Staubli VAL3: sad_proj_sin.dtx

public frame fReference = {x=1365.054, y=-125.975, z=-1150, rz=90, fatherId=world[0]}
public jointRx jPark = {j3=90, j5=90}
public jointRx jJoint = {j1=-39.51779, j2=74.82624, j3=56.29695, j5=48.87681, j6=-167.66375}
public mdesc mNomSpeed = {tmax=100, rmax=100, leave=0.1, reach=0.1, blend=cartesian}
public pointRx pPoint[4564]
  [0] = {x=-1000, z=100, rx=180, rz=141.854, shoulder=lefty, elbow=epositive, wrist=wpositive, fatherId=fReference[0]}
  [1] = {x=-1000, rx=180, rz=141.854, shoulder=lefty, elbow=epositive, wrist=wpositive, fatherId=fReference[0]}
  [2] = {x=-1000, rx=180, rz=141.854, shoulder=lefty, elbow=epositive, wrist=wpositive, fatherId=fReference[0]}
  [3] = {x=-998.763, y=0.971, rx=180, rz=141.854, shoulder=lefty, elbow=epositive, wrist=wpositive, fatherId=fReference[0]}
  [4] = {x=-997.527, y=1.942, rx=180, rz=141.855, shoulder=lefty, elbow=epositive, wrist=wpositive, fatherId=fReference[0]}
  [5] = {x=-996.29, y=2.914, rx=180, rz=141.857, shoulder=lefty, elbow=epositive, wrist=wpositive, fatherId=fReference[0]}
  [6] = {x=-995.054, y=3.885, rx=180, rz=141.858, shoulder=lefty, elbow=epositive, wrist=wpositive, fatherId=fReference[0]}
  [7] = {x=-993.817, y=4.856, rx=180, rz=141.86, shoulder=lefty, elbow=epositive, wrist=wpositive, fatherId=fReference[0]}
  [8] = {x=-992.58, y=5.827, rx=180, rz=141.863, shoulder=lefty, elbow=epositive, wrist=wpositive, fatherId=fReference[0]}
  [9] = {x=-991.344, y=6.798, rx=180, rz=141.866, shoulder=lefty, elbow=epositive, wrist=wpositive, fatherId=fReference[0]}
  [10] = {x=-990.107, y=7.769, rx=180, rz=141.869, shoulder=lefty, elbow=epositive, wrist=wpositive, fatherId=fReference[0]}
  [11] = {x=-988.87, y=8.739, rx=180, rz=141.873, shoulder=lefty, elbow=epositive, wrist=wpositive, fatherId=fReference[0]}
  [12] = {x=-987.634, y=9.71, rx=180, rz=141.877, shoulder=lefty, elbow=epositive, wrist=wpositive, fatherId=fReference[0]}
  [13] = {x=-986.397, y=10.681, rx=180, rz=141.882, shoulder=lefty, elbow=epositive, wrist=wpositive, fatherId=fReference[0]}
  [14] = {x=-985.16, y=11.651, rx=180, rz=141.887, shoulder=lefty, elbow=epositive, wrist=wpositive, fatherId=fReference[0]}
  [15] = {x=-983.923, y=12.622, rx=180, rz=141.892, shoulder=lefty, elbow=epositive, wrist=wpositive, fatherId=fReference[0]}
  [16] = {x=-982.686, y=13.592, rx=180, rz=141.898, shoulder=lefty, elbow=epositive, wrist=wpositive, fatherId=fReference[0]}
  [17] = {x=-981.449, y=14.562, rx=180, rz=141.904, shoulder=lefty, elbow=epositive, wrist=wpositive, fatherId=fReference[0]}
  [18] = {x=-980.211, y=15.532, rx=180, rz=141.911, shoulder=lefty, elbow=epositive, wrist=wpositive, fatherId=fReference[0]}
  [19] = {x=-978.974, y=16.502, rx=180, rz=141.918, shoulder=lefty, elbow=epositive, wrist=wpositive, fatherId=fReference[0]}
  [20] = {x=-977.737, y=17.471, rx=180, rz=141.926, shoulder=lefty, elbow=epositive, wrist=wpositive, fatherId=fReference[0]}
  [21] = {x=-976.499, y=18.441, rx=180, rz=141.934, shoulder=lefty, elbow=epositive, wrist=wpositive, fatherId=fReference[0]}
  [22] = {x=-975.262, y=19.41, rx=180, rz=141.942, shoulder=lefty, elbow=epositive, wrist=wpositive, fatherId=fReference[0]}
  [23] = {x=-974.024, y=20.379, rx=180, rz=141.951, shoulder=lefty, elbow=epositive, wrist=wpositive, fatherId=fReference[0]}
  [24] = {x=-972.786, y=21.347, rx=180, rz=141.96, shoulder=lefty, elbow=epositive, wrist=wpositive, fatherId=fReference[0]}
  [25] = {x=-971.549, y=22.316, rx=180, rz=141.97, shoulder=lefty, elbow=epositive, wrist=wpositive, fatherId=fReference[0]}
  [26] = {x=-970.311, y=23.284, rx=180, rz=141.98, shoulder=lefty, elbow=epositive, wrist=wpositive, fatherId=fReference[0]}
  [27] = {x=-969.072, y=24.252, rx=180, rz=141.991, shoulder=lefty, elbow=epositive, wrist=wpositive, fatherId=fReference[0]}
  [28] = {x=-967.834, y=25.22, rx=180, rz=142.002, shoulder=lefty, elbow=epositive, wrist=wpositive, fatherId=fReference[0]}
  [29] = {x=-966.596, y=26.187, rx=180, rz=142.013, shoulder=lefty, elbow=epositive, wrist=wpositive, fatherId=fReference[0]}
  [30] = {x=-965.357, y=27.155, rx=180, rz=142.025, shoulder=lefty, elbow=epositive, wrist=wpositive, fatherId=fReference[0]}
  [31] = {x=-964.119, y=28.121, rx=180, rz=142.037, shoulder=lefty, elbow=epositive, wrist=wpositive, fatherId=fReference[0]}
  [32] = {x=-962.88, y=29.088, rx=180, rz=142.05, shoulder=lefty, elbow=epositive, wrist=wpositive, fatherId=fReference[0]}
  [33] = {x=-961.641, y=30.054, rx=180, rz=142.063, shoulder=lefty, elbow=epositive, wrist=wpositive, fatherId=fReference[0]}
  [34] = {x=-960.402, y=31.02, rx=180, rz=142.076, shoulder=lefty, elbow=epositive, wrist=wpositive, fatherId=fReference[0]}
  [35] = {x=-959.163, y=31.986, rx=180, rz=142.09, shoulder=lefty, elbow=epositive, wrist=wpositive, fatherId=fReference[0]}
  [36] = {x=-957.923, y=32.951, rx=180, rz=142.105, shoulder=lefty, elbow=epositive, wrist=wpositive, fatherId=fReference[0]}
  [37] = {x=-956.684, y=33.916, rx=180, rz=142.12, shoulder=lefty, elbow=epositive, wrist=wpositive, fatherId=fReference[0]}
  [38] = {x=-955.444, y=34.88, rx=180, rz=142.135, shoulder=lefty, elbow=epositive, wrist=wpositive, fatherId=fReference[0]}
  [39] = {x=-954.204, y=35.844, rx=180, rz=142.151, shoulder=lefty, elbow=epositive, wrist=wpositive, fatherId=fReference[0]}
  [40] = {x=-952.964, y=36.808, rx=180, rz=142.167, shoulder=lefty, elbow=epositive, wrist=wpositive, fatherId=fReference[0]}
  [41] = {x=-951.724, y=37.771, rx=180, rz=142.183, shoulder=lefty, elbow=epositive, wrist=wpositive, fatherId=fReference[0]}
  [42] = {x=-950.483, y=38.734, rx=180, rz=142.2, shoulder=lefty, elbow=epositive, wrist=wpositive, fatherId=fReference[0]}
  [43] = {x=-949.243, y=39.696, rx=180, rz=142.218, shoulder=lefty, elbow=epositive, wrist=wpositive, fatherId=fReference[0]}
  [44] = {x=-948.002, y=40.658, rx=180, rz=142.235, shoulder=lefty, elbow=epositive, wrist=wpositive, fatherId=fReference[0]}
  [45] = {x=-946.761, y=41.619, rx=180, rz=142.254, shoulder=lefty, elbow=epositive, wrist=wpositive, fatherId=fReference[0]}
  [46] = {x=-945.52, y=42.58, rx=180, rz=142.272, shoulder=lefty, elbow=epositive, wrist=wpositive, fatherId=fReference[0]}
  [47] = {x=-944.278, y=43.541, rx=180, rz=142.291, shoulder=lefty, elbow=epositive, wrist=wpositive, fatherId=fReference[0]}
  [48] = {x=-943.037, y=44.501, rx=180, rz=142.311, shoulder=lefty, elbow=epositive, wrist=wpositive, fatherId=fReference[0]}
  [49] = {x=-941.795, y=45.46, rx=180, rz=142.331, shoulder=lefty, elbow=epositive, wrist=wpositive, fatherId=fReference[0]}
  [50] = {x=-940.553, y=46.419, rx=180, rz=142.351, shoulder=lefty, elbow=epositive, wrist=wpositive, fatherId=fReference[0]}
  [51] = {x=-939.31, y=47.377, rx=180, rz=142.372, shoulder=lefty, elbow=epositive, wrist=wpositive, fatherId=fReference[0]}
  [52] = {x=-938.068, y=48.335, rx=180, rz=142.394, shoulder=lefty, elbow=epositive, wrist=wpositive, fatherId=fReference[0]}
  [53] = {x=-936.825, y=49.292, rx=180, rz=142.415, shoulder=lefty, elbow=epositive, wrist=wpositive, fatherId=fReference[0]}
  [54] = {x=-935.582, y=50.249, rx=180, rz=142.438, shoulder=lefty, elbow=epositive, wrist=wpositive, fatherId=fReference[0]}
  [55] = {x=-934.339, y=51.205, rx=180, rz=142.46, shoulder=lefty, elbow=epositive, wrist=wpositive, fatherId=fReference[0]}
  [56] = {x=-933.095, y=52.161, rx=180, rz=142.483, shoulder=lefty, elbow=epositive, wrist=wpositive, fatherId=fReference[0]}
  [57] = {x=-931.852, y=53.116, rx=180, rz=142.507, shoulder=lefty, elbow=epositive, wrist=wpositive, fatherId=fReference[0]}
  [58] = {x=-930.608, y=54.07, rx=180, rz=142.531, shoulder=lefty, elbow=epositive, wrist=wpositive, fatherId=fReference[0]}
  [59] = {x=-929.363, y=55.024, rx=180, rz=142.555, shoulder=lefty, elbow=epositive, wrist=wpositive, fatherId=fReference[0]}
  [60] = {x=-928.119, y=55.977, rx=180, rz=142.58, shoulder=lefty, elbow=epositive, wrist=wpositive, fatherId=fReference[0]}
  [61] = {x=-926.874, y=56.929, rx=180, rz=142.605, shoulder=lefty, elbow=epositive, wrist=wpositive, fatherId=fReference[0]}
  [62] = {x=-925.629, y=57.881, rx=180, rz=142.631, shoulder=lefty, elbow=epositive, wrist=wpositive, fatherId=fReference[0]}
  [63] = {x=-924.384, y=58.832, rx=180, rz=142.657, shoulder=lefty, elbow=epositive, wrist=wpositive, fatherId=fReference[0]}
  [64] = {x=-923.138, y=59.782, rx=180, rz=142.684, shoulder=lefty, elbow=epositive, wrist=wpositive, fatherId=fReference[0]}
  [65] = {x=-921.892, y=60.732, rx=180, rz=142.711, shoulder=lefty, elbow=epositive, wrist=wpositive, fatherId=fReference[0]}
  [66] = {x=-920.646, y=61.681, rx=180, rz=142.738, shoulder=lefty, elbow=epositive, wrist=wpositive, fatherId=fReference[0]}
  [67] = {x=-919.4, y=62.629, rx=180, rz=142.766, shoulder=lefty, elbow=epositive, wrist=wpositive, fatherId=fReference[0]}
  [68] = {x=-918.153, y=63.576, rx=180, rz=142.795, shoulder=lefty, elbow=epositive, wrist=wpositive, fatherId=fReference[0]}
  [69] = {x=-916.906, y=64.523, rx=180, rz=142.824, shoulder=lefty, elbow=epositive, wrist=wpositive, fatherId=fReference[0]}
  [70] = {x=-915.659, y=65.469, rx=180, rz=142.853, shoulder=lefty, elbow=epositive, wrist=wpositive, fatherId=fReference[0]}
  [71] = {x=-914.411, y=66.414, rx=180, rz=142.883, shoulder=lefty, elbow=epositive, wrist=wpositive, fatherId=fReference[0]}
  [72] = {x=-913.163, y=67.358, rx=180, rz=142.913, shoulder=lefty, elbow=epositive, wrist=wpositive, fatherId=fReference[0]}
  [73] = {x=-911.915, y=68.302, rx=180, rz=142.944, shoulder=lefty, elbow=epositive, wrist=wpositive, fatherId=fReference[0]}
  [74] = {x=-910.667, y=69.245, rx=180, rz=142.975, shoulder=lefty, elbow=epositive, wrist=wpositive, fatherId=fReference[0]}
  [75] = {x=-909.418, y=70.187, rx=180, rz=143.007, shoulder=lefty, elbow=epositive, wrist=wpositive, fatherId=fReference[0]}
  [76] = {x=-908.169, y=71.128, rx=180, rz=143.039, shoulder=lefty, elbow=epositive, wrist=wpositive, fatherId=fReference[0]}
  [77] = {x=-906.919, y=72.068, rx=180, rz=143.071, shoulder=lefty, elbow=epositive, wrist=wpositive, fatherId=fReference[0]}
  [78] = {x=-905.67, y=73.007, rx=180, rz=143.104, shoulder=lefty, elbow=epositive, wrist=wpositive, fatherId=fReference[0]}
  [79] = {x=-904.419, y=73.946, rx=180, rz=143.138, shoulder=lefty, elbow=epositive, wrist=wpositive, fatherId=fReference[0]}
  [80] = {x=-903.169, y=74.883, rx=180, rz=143.172, shoulder=lefty, elbow=epositive, wrist=wpositive, fatherId=fReference[0]}
  [81] = {x=-901.918, y=75.82, rx=180, rz=143.206, shoulder=lefty, elbow=epositive, wrist=wpositive, fatherId=fReference[0]}
  [82] = {x=-900.667, y=76.756, rx=180, rz=143.241, shoulder=lefty, elbow=epositive, wrist=wpositive, fatherId=fReference[0]}
  [83] = {x=-899.416, y=77.691, rx=180, rz=143.276, shoulder=lefty, elbow=epositive, wrist=wpositive, fatherId=fReference[0]}
  [84] = {x=-898.164, y=78.625, rx=180, rz=143.312, shoulder=lefty, elbow=epositive, wrist=wpositive, fatherId=fReference[0]}
  [85] = {x=-896.912, y=79.557, rx=180, rz=143.348, shoulder=lefty, elbow=epositive, wrist=wpositive, fatherId=fReference[0]}
  [86] = {x=-895.659, y=80.489, rx=180, rz=143.385, shoulder=lefty, elbow=epositive, wrist=wpositive, fatherId=fReference[0]}
  [87] = {x=-894.406, y=81.42, rx=180, rz=143.422, shoulder=lefty, elbow=epositive, wrist=wpositive, fatherId=fReference[0]}
  [88] = {x=-893.153, y=82.35, rx=180, rz=143.46, shoulder=lefty, elbow=epositive, wrist=wpositive, fatherId=fReference[0]}
  [89] = {x=-891.899, y=83.279, rx=180, rz=143.498, shoulder=lefty, elbow=epositive, wrist=wpositive, fatherId=fReference[0]}
  [90] = {x=-890.645, y=84.207, rx=180, rz=143.536, shoulder=lefty, elbow=epositive, wrist=wpositive, fatherId=fReference[0]}
  [91] = {x=-889.391, y=85.134, rx=180, rz=143.575, shoulder=lefty, elbow=epositive, wrist=wpositive, fatherId=fReference[0]}
  [92] = {x=-888.136, y=86.06, rx=180, rz=143.615, shoulder=lefty, elbow=epositive, wrist=wpositive, fatherId=fReference[0]}
  [93] = {x=-886.881, y=86.985, rx=180, rz=143.655, shoulder=lefty, elbow=epositive, wrist=wpositive, fatherId=fReference[0]}
  [94] = {x=-885.626, y=87.909, rx=180, rz=143.696, shoulder=lefty, elbow=epositive, wrist=wpositive, fatherId=fReference[0]}
  [95] = {x=-884.37, y=88.832, rx=180, rz=143.737, shoulder=lefty, elbow=epositive, wrist=wpositive, fatherId=fReference[0]}
  [96] = {x=-883.113, y=89.753, rx=180, rz=143.778, shoulder=lefty, elbow=epositive, wrist=wpositive, fatherId=fReference[0]}
  [97] = {x=-881.857, y=90.674, rx=180, rz=143.82, shoulder=lefty, elbow=epositive, wrist=wpositive, fatherId=fReference[0]}
  [98] = {x=-880.6, y=91.593, rx=180, rz=143.862, shoulder=lefty, elbow=epositive, wrist=wpositive, fatherId=fReference[0]}
  [99] = {x=-879.342, y=92.511, rx=180, rz=143.905, shoulder=lefty, elbow=epositive, wrist=wpositive, fatherId=fReference[0]}
  [100] = {x=-878.084, y=93.428, rx=180, rz=143.949, shoulder=lefty, elbow=epositive, wrist=wpositive, fatherId=fReference[0]}
  [101] = {x=-876.826, y=94.344, rx=180, rz=143.993, shoulder=lefty, elbow=epositive, wrist=wpositive, fatherId=fReference[0]}
  [102] = {x=-875.567, y=95.259, rx=180, rz=144.037, shoulder=lefty, elbow=epositive, wrist=wpositive, fatherId=fReference[0]}
  [103] = {x=-874.308, y=96.173, rx=180, rz=144.082, shoulder=lefty, elbow=epositive, wrist=wpositive, fatherId=fReference[0]}
  [104] = {x=-873.049, y=97.085, rx=180, rz=144.127, shoulder=lefty, elbow=epositive, wrist=wpositive, fatherId=fReference[0]}
  [105] = {x=-871.789, y=97.996, rx=180, rz=144.173, shoulder=lefty, elbow=epositive, wrist=wpositive, fatherId=fReference[0]}
  [106] = {x=-870.528, y=98.906, rx=180, rz=144.22, shoulder=lefty, elbow=epositive, wrist=wpositive, fatherId=fReference[0]}
  [107] = {x=-869.267, y=99.815, rx=180, rz=144.266, shoulder=lefty, elbow=epositive, wrist=wpositive, fatherId=fReference[0]}
  [108] = {x=-868.006, y=100.722, rx=180, rz=144.314, shoulder=lefty, elbow=epositive, wrist=wpositive, fatherId=fReference[0]}
  [109] = {x=-866.745, y=101.628, rx=180, rz=144.362, shoulder=lefty, elbow=epositive, wrist=wpositive, fatherId=fReference[0]}
  [110] = {x=-865.482, y=102.533, rx=180, rz=144.41, shoulder=lefty, elbow=epositive, wrist=wpositive, fatherId=fReference[0]}
  [111] = {x=-864.22, y=103.437, rx=180, rz=144.459, shoulder=lefty, elbow=epositive, wrist=wpositive, fatherId=fReference[0]}
  [112] = {x=-862.957, y=104.339, rx=180, rz=144.508, shoulder=lefty, elbow=epositive, wrist=wpositive, fatherId=fReference[0]}
  [113] = {x=-861.693, y=105.24, rx=180, rz=144.558, shoulder=lefty, elbow=epositive, wrist=wpositive, fatherId=fReference[0]}
  [114] = {x=-860.429, y=106.139, rx=180, rz=144.609, shoulder=lefty, elbow=epositive, wrist=wpositive, fatherId=fReference[0]}
  [115] = {x=-859.165, y=107.038, rx=180, rz=144.659, shoulder=lefty, elbow=epositive, wrist=wpositive, fatherId=fReference[0]}
  [116] = {x=-857.9, y=107.935, rx=180, rz=144.711, shoulder=lefty, elbow=epositive, wrist=wpositive, fatherId=fReference[0]}
  [117] = {x=-856.635, y=108.83, rx=180, rz=144.763, shoulder=lefty, elbow=epositive, wrist=wpositive, fatherId=fReference[0]}
  [118] = {x=-855.369, y=109.724, rx=180, rz=144.815, shoulder=lefty, elbow=epositive, wrist=wpositive, fatherId=fReference[0]}
  [119] = {x=-854.103, y=110.617, rx=180, rz=144.868, shoulder=lefty, elbow=epositive, wrist=wpositive, fatherId=fReference[0]}
  [120] = {x=-852.836, y=111.508, rx=180, rz=144.922, shoulder=lefty, elbow=epositive, wrist=wpositive, fatherId=fReference[0]}
  [121] = {x=-851.569, y=112.398, rx=180, rz=144.976, shoulder=lefty, elbow=epositive, wrist=wpositive, fatherId=fReference[0]}
  [122] = {x=-850.301, y=113.287, rx=180, rz=145.03, shoulder=lefty, elbow=epositive, wrist=wpositive, fatherId=fReference[0]}
  [123] = {x=-849.033, y=114.174, rx=180, rz=145.085, shoulder=lefty, elbow=epositive, wrist=wpositive, fatherId=fReference[0]}
  [124] = {x=-847.764, y=115.059, rx=180, rz=145.141, shoulder=lefty, elbow=epositive, wrist=wpositive, fatherId=fReference[0]}
  [125] = {x=-846.495, y=115.943, rx=180, rz=145.197, shoulder=lefty, elbow=epositive, wrist=wpositive, fatherId=fReference[0]}
  [126] = {x=-845.225, y=116.826, rx=180, rz=145.253, shoulder=lefty, elbow=epositive, wrist=wpositive, fatherId=fReference[0]}
  [127] = {x=-843.955, y=117.707, rx=180, rz=145.311, shoulder=lefty, elbow=epositive, wrist=wpositive, fatherId=fReference[0]}
  [128] = {x=-842.685, y=118.586, rx=180, rz=145.368, shoulder=lefty, elbow=epositive, wrist=wpositive, fatherId=fReference[0]}
  [129] = {x=-841.413, y=119.464, rx=-180, rz=145.426, shoulder=lefty, elbow=epositive, wrist=wpositive, fatherId=fReference[0]}
  [130] = {x=-840.142, y=120.341, rx=180, rz=145.485, shoulder=lefty, elbow=epositive, wrist=wpositive, fatherId=fReference[0]}
  [131] = {x=-838.869, y=121.216, rx=180, rz=145.544, shoulder=lefty, elbow=epositive, wrist=wpositive, fatherId=fReference[0]}
  [132] = {x=-837.597, y=122.089, rx=180, rz=145.604, shoulder=lefty, elbow=epositive, wrist=wpositive, fatherId=fReference[0]}
  [133] = {x=-836.323, y=122.961, rx=180, rz=145.665, shoulder=lefty, elbow=epositive, wrist=wpositive, fatherId=fReference[0]}
  [134] = {x=-835.049, y=123.831, rx=180, rz=145.725, shoulder=lefty, elbow=epositive, wrist=wpositive, fatherId=fReference[0]}
  [135] = {x=-833.775, y=124.699, rx=180, rz=145.787, shoulder=lefty, elbow=epositive, wrist=wpositive, fatherId=fReference[0]}
  [136] = {x=-832.5, y=125.566, rx=180, rz=145.849, shoulder=lefty, elbow=epositive, wrist=wpositive, fatherId=fReference[0]}
  [137] = {x=-831.225, y=126.431, rx=180, rz=145.911, shoulder=lefty, elbow=epositive, wrist=wpositive, fatherId=fReference[0]}
  [138] = {x=-829.949, y=127.295, rx=180, rz=145.974, shoulder=lefty, elbow=epositive, wrist=wpositive, fatherId=fReference[0]}
  [139] = {x=-828.672, y=128.157, rx=180, rz=146.038, shoulder=lefty, elbow=epositive, wrist=wpositive, fatherId=fReference[0]}
  [140] = {x=-827.395, y=129.017, rx=180, rz=146.102, shoulder=lefty, elbow=epositive, wrist=wpositive, fatherId=fReference[0]}
  [141] = {x=-826.117, y=129.876, rx=180, rz=146.167, shoulder=lefty, elbow=epositive, wrist=wpositive, fatherId=fReference[0]}
  [142] = {x=-824.839, y=130.732, rx=180, rz=146.232, shoulder=lefty, elbow=epositive, wrist=wpositive, fatherId=fReference[0]}
  [143] = {x=-823.56, y=131.587, rx=180, rz=146.298, shoulder=lefty, elbow=epositive, wrist=wpositive, fatherId=fReference[0]}
  [144] = {x=-822.281, y=132.441, rx=180, rz=146.364, shoulder=lefty, elbow=epositive, wrist=wpositive, fatherId=fReference[0]}
  [145] = {x=-821.001, y=133.292, rx=180, rz=146.431, shoulder=lefty, elbow=epositive, wrist=wpositive, fatherId=fReference[0]}
  [146] = {x=-819.721, y=134.142, rx=180, rz=146.499, shoulder=lefty, elbow=epositive, wrist=wpositive, fatherId=fReference[0]}
  [147] = {x=-818.44, y=134.99, rx=180, rz=146.567, shoulder=lefty, elbow=epositive, wrist=wpositive, fatherId=fReference[0]}
  [148] = {x=-817.158, y=135.836, rx=180, rz=146.636, shoulder=lefty, elbow=epositive, wrist=wpositive, fatherId=fReference[0]}
  [149] = {x=-815.876, y=136.68, rx=180, rz=146.705, shoulder=lefty, elbow=epositive, wrist=wpositive, fatherId=fReference[0]}
  [150] = {x=-814.593, y=137.523, rx=180, rz=146.775, shoulder=lefty, elbow=epositive, wrist=wpositive, fatherId=fReference[0]}
  [151] = {x=-813.309, y=138.364, rx=180, rz=146.845, shoulder=lefty, elbow=epositive, wrist=wpositive, fatherId=fReference[0]}
  [152] = {x=-812.025, y=139.202, rx=180, rz=146.916, shoulder=lefty, elbow=epositive, wrist=wpositive, fatherId=fReference[0]}
  [153] = {x=-810.74, y=140.039, rx=180, rz=146.987, shoulder=lefty, elbow=epositive, wrist=wpositive, fatherId=fReference[0]}
  [154] = {x=-809.455, y=140.875, rx=180, rz=147.059, shoulder=lefty, elbow=epositive, wrist=wpositive, fatherId=fReference[0]}
  [155] = {x=-808.169, y=141.708, rx=180, rz=147.132, shoulder=lefty, elbow=epositive, wrist=wpositive, fatherId=fReference[0]}
  [156] = {x=-806.883, y=142.539, rx=180, rz=147.205, shoulder=lefty, elbow=epositive, wrist=wpositive, fatherId=fReference[0]}
  [157] = {x=-805.596, y=143.368, rx=180, rz=147.279, shoulder=lefty, elbow=epositive, wrist=wpositive, fatherId=fReference[0]}
  [158] = {x=-804.308, y=144.196, rx=180, rz=147.353, shoulder=lefty, elbow=epositive, wrist=wpositive, fatherId=fReference[0]}
  [159] = {x=-803.019, y=145.021, rx=180, rz=147.428, shoulder=lefty, elbow=epositive, wrist=wpositive, fatherId=fReference[0]}
  [160] = {x=-801.73, y=145.845, rx=180, rz=147.504, shoulder=lefty, elbow=epositive, wrist=wpositive, fatherId=fReference[0]}
  [161] = {x=-800.44, y=146.666, rx=180, rz=147.58, shoulder=lefty, elbow=epositive, wrist=wpositive, fatherId=fReference[0]}
  [162] = {x=-799.15, y=147.486, rx=180, rz=147.657, shoulder=lefty, elbow=epositive, wrist=wpositive, fatherId=fReference[0]}
  [163] = {x=-797.859, y=148.303, rx=180, rz=147.734, shoulder=lefty, elbow=epositive, wrist=wpositive, fatherId=fReference[0]}
  [164] = {x=-796.567, y=149.119, rx=180, rz=147.812, shoulder=lefty, elbow=epositive, wrist=wpositive, fatherId=fReference[0]}
  [165] = {x=-795.275, y=149.932, rx=-180, rz=147.891, shoulder=lefty, elbow=epositive, wrist=wpositive, fatherId=fReference[0]}
  [166] = {x=-793.982, y=150.744, rx=180, rz=147.97, shoulder=lefty, elbow=epositive, wrist=wpositive, fatherId=fReference[0]}
  [167] = {x=-792.688, y=151.553, rx=180, rz=148.05, shoulder=lefty, elbow=epositive, wrist=wpositive, fatherId=fReference[0]}
  [168] = {x=-791.394, y=152.36, rx=180, rz=148.13, shoulder=lefty, elbow=epositive, wrist=wpositive, fatherId=fReference[0]}
  [169] = {x=-790.099, y=153.165, rx=180, rz=148.211, shoulder=lefty, elbow=epositive, wrist=wpositive, fatherId=fReference[0]}
  [170] = {x=-788.803, y=153.968, rx=180, rz=148.293, shoulder=lefty, elbow=epositive, wrist=wpositive, fatherId=fReference[0]}
  [171] = {x=-787.507, y=154.769, rx=180, rz=148.375, shoulder=lefty, elbow=epositive, wrist=wpositive, fatherId=fReference[0]}
  [172] = {x=-786.21, y=155.568, rx=180, rz=148.458, shoulder=lefty, elbow=epositive, wrist=wpositive, fatherId=fReference[0]}
  [173] = {x=-784.912, y=156.365, rx=-180, rz=148.541, shoulder=lefty, elbow=epositive, wrist=wpositive, fatherId=fReference[0]}
  [174] = {x=-783.613, y=157.159, rx=180, rz=148.625, shoulder=lefty, elbow=epositive, wrist=wpositive, fatherId=fReference[0]}
  [175] = {x=-782.314, y=157.951, rx=180, rz=148.71, shoulder=lefty, elbow=epositive, wrist=wpositive, fatherId=fReference[0]}
  [176] = {x=-781.014, y=158.741, rx=180, rz=148.795, shoulder=lefty, elbow=epositive, wrist=wpositive, fatherId=fReference[0]}
  [177] = {x=-779.714, y=159.529, rx=180, rz=148.881, shoulder=lefty, elbow=epositive, wrist=wpositive, fatherId=fReference[0]}
  [178] = {x=-778.413, y=160.315, rx=180, rz=148.968, shoulder=lefty, elbow=epositive, wrist=wpositive, fatherId=fReference[0]}
  [179] = {x=-777.111, y=161.098, rx=180, rz=149.055, shoulder=lefty, elbow=epositive, wrist=wpositive, fatherId=fReference[0]}
  [180] = {x=-775.808, y=161.879, rx=180, rz=149.143, shoulder=lefty, elbow=epositive, wrist=wpositive, fatherId=fReference[0]}
  [181] = {x=-774.505, y=162.658, rx=180, rz=149.231, shoulder=lefty, elbow=epositive, wrist=wpositive, fatherId=fReference[0]}
  [182] = {x=-773.2, y=163.434, rx=180, rz=149.32, shoulder=lefty, elbow=epositive, wrist=wpositive, fatherId=fReference[0]}
  [183] = {x=-771.896, y=164.208, rx=180, rz=149.41, shoulder=lefty, elbow=epositive, wrist=wpositive, fatherId=fReference[0]}
  [184] = {x=-770.59, y=164.98, rx=180, rz=149.5, shoulder=lefty, elbow=epositive, wrist=wpositive, fatherId=fReference[0]}
  [185] = {x=-769.284, y=165.75, rx=180, rz=149.591, shoulder=lefty, elbow=epositive, wrist=wpositive, fatherId=fReference[0]}
  [186] = {x=-767.977, y=166.517, rx=180, rz=149.683, shoulder=lefty, elbow=epositive, wrist=wpositive, fatherId=fReference[0]}
  [187] = {x=-766.669, y=167.281, rx=180, rz=149.775, shoulder=lefty, elbow=epositive, wrist=wpositive, fatherId=fReference[0]}
  [188] = {x=-765.36, y=168.044, rx=180, rz=149.868, shoulder=lefty, elbow=epositive, wrist=wpositive, fatherId=fReference[0]}
  [189] = {x=-764.051, y=168.804, rx=180, rz=149.962, shoulder=lefty, elbow=epositive, wrist=wpositive, fatherId=fReference[0]}
  [190] = {x=-762.741, y=169.561, rx=180, rz=150.056, shoulder=lefty, elbow=epositive, wrist=wpositive, fatherId=fReference[0]}
  [191] = {x=-761.431, y=170.316, rx=180, rz=150.151, shoulder=lefty, elbow=epositive, wrist=wpositive, fatherId=fReference[0]}
  [192] = {x=-760.119, y=171.069, rx=180, rz=150.247, shoulder=lefty, elbow=epositive, wrist=wpositive, fatherId=fReference[0]}
  [193] = {x=-758.807, y=171.819, rx=180, rz=150.343, shoulder=lefty, elbow=epositive, wrist=wpositive, fatherId=fReference[0]}
  [194] = {x=-757.494, y=172.566, rx=180, rz=150.44, shoulder=lefty, elbow=epositive, wrist=wpositive, fatherId=fReference[0]}
  [195] = {x=-756.181, y=173.311, rx=180, rz=150.537, shoulder=lefty, elbow=epositive, wrist=wpositive, fatherId=fReference[0]}
  [196] = {x=-754.866, y=174.054, rx=180, rz=150.636, shoulder=lefty, elbow=epositive, wrist=wpositive, fatherId=fReference[0]}
  [197] = {x=-753.551, y=174.794, rx=180, rz=150.734, shoulder=lefty, elbow=epositive, wrist=wpositive, fatherId=fReference[0]}
  [198] = {x=-752.235, y=175.531, rx=-180, rz=150.834, shoulder=lefty, elbow=epositive, wrist=wpositive, fatherId=fReference[0]}
  [199] = {x=-750.919, y=176.266, rx=-180, rz=150.934, shoulder=lefty, elbow=epositive, wrist=wpositive, fatherId=fReference[0]}
  [200] = {x=-749.601, y=176.998, rx=-180, rz=151.035, shoulder=lefty, elbow=epositive, wrist=wpositive, fatherId=fReference[0]}
  [201] = {x=-748.283, y=177.727, rx=180, rz=151.137, shoulder=lefty, elbow=epositive, wrist=wpositive, fatherId=fReference[0]}
  [202] = {x=-746.965, y=178.454, rx=180, rz=151.239, shoulder=lefty, elbow=epositive, wrist=wpositive, fatherId=fReference[0]}
  [203] = {x=-745.645, y=179.179, rx=180, rz=151.342, shoulder=lefty, elbow=epositive, wrist=wpositive, fatherId=fReference[0]}
  [204] = {x=-744.325, y=179.9, rx=180, rz=151.445, shoulder=lefty, elbow=epositive, wrist=wpositive, fatherId=fReference[0]}
  [205] = {x=-743.004, y=180.619, rx=180, rz=151.549, shoulder=lefty, elbow=epositive, wrist=wpositive, fatherId=fReference[0]}
  [206] = {x=-741.682, y=181.335, rx=180, rz=151.654, shoulder=lefty, elbow=epositive, wrist=wpositive, fatherId=fReference[0]}
  [207] = {x=-740.359, y=182.049, rx=180, rz=151.76, shoulder=lefty, elbow=epositive, wrist=wpositive, fatherId=fReference[0]}
  [208] = {x=-739.036, y=182.76, rx=180, rz=151.866, shoulder=lefty, elbow=epositive, wrist=wpositive, fatherId=fReference[0]}
  [209] = {x=-737.712, y=183.468, rx=180, rz=151.973, shoulder=lefty, elbow=epositive, wrist=wpositive, fatherId=fReference[0]}
  [210] = {x=-736.387, y=184.173, rx=180, rz=152.081, shoulder=lefty, elbow=epositive, wrist=wpositive, fatherId=fReference[0]}
  [211] = {x=-735.061, y=184.875, rx=180, rz=152.189, shoulder=lefty, elbow=epositive, wrist=wpositive, fatherId=fReference[0]}
  [212] = {x=-733.735, y=185.575, rx=180, rz=152.298, shoulder=lefty, elbow=epositive, wrist=wpositive, fatherId=fReference[0]}
  [213] = {x=-732.408, y=186.272, rx=180, rz=152.408, shoulder=lefty, elbow=epositive, wrist=wpositive, fatherId=fReference[0]}
  [214] = {x=-731.08, y=186.966, rx=-180, rz=152.518, shoulder=lefty, elbow=epositive, wrist=wpositive, fatherId=fReference[0]}
  [215] = {x=-729.751, y=187.657, rx=180, rz=152.63, shoulder=lefty, elbow=epositive, wrist=wpositive, fatherId=fReference[0]}
  [216] = {x=-728.422, y=188.345, rx=180, rz=152.741, shoulder=lefty, elbow=epositive, wrist=wpositive, fatherId=fReference[0]}
  [217] = {x=-727.092, y=189.03, rx=180, rz=152.854, shoulder=lefty, elbow=epositive, wrist=wpositive, fatherId=fReference[0]}
  [218] = {x=-725.761, y=189.713, rx=180, rz=152.967, shoulder=lefty, elbow=epositive, wrist=wpositive, fatherId=fReference[0]}
  [219] = {x=-724.429, y=190.392, rx=180, rz=153.081, shoulder=lefty, elbow=epositive, wrist=wpositive, fatherId=fReference[0]}
  [220] = {x=-723.097, y=191.069, rx=180, rz=153.196, shoulder=lefty, elbow=epositive, wrist=wpositive, fatherId=fReference[0]}
  [221] = {x=-721.764, y=191.742, rx=180, rz=153.311, shoulder=lefty, elbow=epositive, wrist=wpositive, fatherId=fReference[0]}
  [222] = {x=-720.43, y=192.413, rx=180, rz=153.427, shoulder=lefty, elbow=epositive, wrist=wpositive, fatherId=fReference[0]}
  [223] = {x=-719.095, y=193.08, rx=180, rz=153.544, shoulder=lefty, elbow=epositive, wrist=wpositive, fatherId=fReference[0]}
  [224] = {x=-717.76, y=193.745, rx=180, rz=153.661, shoulder=lefty, elbow=epositive, wrist=wpositive, fatherId=fReference[0]}
  [225] = {x=-716.424, y=194.406, rx=-180, rz=153.779, shoulder=lefty, elbow=epositive, wrist=wpositive, fatherId=fReference[0]}
  [226] = {x=-715.087, y=195.065, rx=180, rz=153.898, shoulder=lefty, elbow=epositive, wrist=wpositive, fatherId=fReference[0]}
  [227] = {x=-713.749, y=195.72, rx=180, rz=154.017, shoulder=lefty, elbow=epositive, wrist=wpositive, fatherId=fReference[0]}
  [228] = {x=-712.411, y=196.372, rx=180, rz=154.138, shoulder=lefty, elbow=epositive, wrist=wpositive, fatherId=fReference[0]}
  [229] = {x=-711.072, y=197.022, rx=180, rz=154.259, shoulder=lefty, elbow=epositive, wrist=wpositive, fatherId=fReference[0]}
  [230] = {x=-709.732, y=197.668, rx=180, rz=154.38, shoulder=lefty, elbow=epositive, wrist=wpositive, fatherId=fReference[0]}
  [231] = {x=-708.391, y=198.311, rx=180, rz=154.503, shoulder=lefty, elbow=epositive, wrist=wpositive, fatherId=fReference[0]}
  [232] = {x=-707.05, y=198.95, rx=180, rz=154.626, shoulder=lefty, elbow=epositive, wrist=wpositive, fatherId=fReference[0]}
  [233] = {x=-705.708, y=199.587, rx=180, rz=154.75, shoulder=lefty, elbow=epositive, wrist=wpositive, fatherId=fReference[0]}
  [234] = {x=-704.365, y=200.22, rx=-180, rz=154.874, shoulder=lefty, elbow=epositive, wrist=wpositive, fatherId=fReference[0]}
  [235] = {x=-703.021, y=200.85, rx=180, rz=154.999, shoulder=lefty, elbow=epositive, wrist=wpositive, fatherId=fReference[0]}
  [236] = {x=-701.677, y=201.477, rx=180, rz=155.125, shoulder=lefty, elbow=epositive, wrist=wpositive, fatherId=fReference[0]}
  [237] = {x=-700.332, y=202.101, rx=180, rz=155.252, shoulder=lefty, elbow=epositive, wrist=wpositive, fatherId=fReference[0]}
  [238] = {x=-698.986, y=202.721, rx=180, rz=155.379, shoulder=lefty, elbow=epositive, wrist=wpositive, fatherId=fReference[0]}
  [239] = {x=-697.639, y=203.338, rx=-180, rz=155.508, shoulder=lefty, elbow=epositive, wrist=wpositive, fatherId=fReference[0]}
  [240] = {x=-696.292, y=203.952, rx=180, rz=155.636, shoulder=lefty, elbow=epositive, wrist=wpositive, fatherId=fReference[0]}
  [241] = {x=-694.944, y=204.563, rx=180, rz=155.766, shoulder=lefty, elbow=epositive, wrist=wpositive, fatherId=fReference[0]}
  [242] = {x=-693.595, y=205.17, rx=-180, rz=155.896, shoulder=lefty, elbow=epositive, wrist=wpositive, fatherId=fReference[0]}
  [243] = {x=-692.246, y=205.774, rx=-180, rz=156.027, shoulder=lefty, elbow=epositive, wrist=wpositive, fatherId=fReference[0]}
  [244] = {x=-690.895, y=206.374, rx=180, rz=156.159, shoulder=lefty, elbow=epositive, wrist=wpositive, fatherId=fReference[0]}
  [245] = {x=-689.544, y=206.971, rx=180, rz=156.291, shoulder=lefty, elbow=epositive, wrist=wpositive, fatherId=fReference[0]}
  [246] = {x=-688.193, y=207.565, rx=180, rz=156.425, shoulder=lefty, elbow=epositive, wrist=wpositive, fatherId=fReference[0]}
  [247] = {x=-686.84, y=208.155, rx=180, rz=156.559, shoulder=lefty, elbow=epositive, wrist=wpositive, fatherId=fReference[0]}
  [248] = {x=-685.487, y=208.741, rx=180, rz=156.693, shoulder=lefty, elbow=epositive, wrist=wpositive, fatherId=fReference[0]}
  [249] = {x=-684.133, y=209.325, rx=180, rz=156.828, shoulder=lefty, elbow=epositive, wrist=wpositive, fatherId=fReference[0]}
  [250] = {x=-682.778, y=209.905, rx=180, rz=156.965, shoulder=lefty, elbow=epositive, wrist=wpositive, fatherId=fReference[0]}
  [251] = {x=-681.423, y=210.481, rx=180, rz=157.101, shoulder=lefty, elbow=epositive, wrist=wpositive, fatherId=fReference[0]}
  [252] = {x=-680.067, y=211.054, rx=180, rz=157.239, shoulder=lefty, elbow=epositive, wrist=wpositive, fatherId=fReference[0]}
  [253] = {x=-678.71, y=211.623, rx=180, rz=157.377, shoulder=lefty, elbow=epositive, wrist=wpositive, fatherId=fReference[0]}
  [254] = {x=-677.353, y=212.189, rx=180, rz=157.516, shoulder=lefty, elbow=epositive, wrist=wpositive, fatherId=fReference[0]}
  [255] = {x=-675.994, y=212.751, rx=180, rz=157.656, shoulder=lefty, elbow=epositive, wrist=wpositive, fatherId=fReference[0]}
  [256] = {x=-674.635, y=213.309, rx=180, rz=157.796, shoulder=lefty, elbow=epositive, wrist=wpositive, fatherId=fReference[0]}
  [257] = {x=-673.276, y=213.864, rx=180, rz=157.937, shoulder=lefty, elbow=epositive, wrist=wpositive, fatherId=fReference[0]}
  [258] = {x=-671.915, y=214.416, rx=180, rz=158.079, shoulder=lefty, elbow=epositive, wrist=wpositive, fatherId=fReference[0]}
  [259] = {x=-670.554, y=214.963, rx=180, rz=158.222, shoulder=lefty, elbow=epositive, wrist=wpositive, fatherId=fReference[0]}
  [260] = {x=-669.193, y=215.508, rx=180, rz=158.365, shoulder=lefty, elbow=epositive, wrist=wpositive, fatherId=fReference[0]}
  [261] = {x=-667.83, y=216.048, rx=180, rz=158.509, shoulder=lefty, elbow=epositive, wrist=wpositive, fatherId=fReference[0]}
  [262] = {x=-666.467, y=216.585, rx=180, rz=158.654, shoulder=lefty, elbow=epositive, wrist=wpositive, fatherId=fReference[0]}
  [263] = {x=-665.103, y=217.118, rx=180, rz=158.799, shoulder=lefty, elbow=epositive, wrist=wpositive, fatherId=fReference[0]}
  [264] = {x=-663.739, y=217.647, rx=180, rz=158.945, shoulder=lefty, elbow=epositive, wrist=wpositive, fatherId=fReference[0]}
  [265] = {x=-662.373, y=218.173, rx=180, rz=159.092, shoulder=lefty, elbow=epositive, wrist=wpositive, fatherId=fReference[0]}
  [266] = {x=-661.007, y=218.694, rx=180, rz=159.24, shoulder=lefty, elbow=epositive, wrist=wpositive, fatherId=fReference[0]}
  [267] = {x=-659.641, y=219.212, rx=180, rz=159.388, shoulder=lefty, elbow=epositive, wrist=wpositive, fatherId=fReference[0]}
  [268] = {x=-658.273, y=219.727, rx=180, rz=159.537, shoulder=lefty, elbow=epositive, wrist=wpositive, fatherId=fReference[0]}
  [269] = {x=-656.905, y=220.237, rx=-180, rz=159.687, shoulder=lefty, elbow=epositive, wrist=wpositive, fatherId=fReference[0]}
  [270] = {x=-655.537, y=220.744, rx=180, rz=159.837, shoulder=lefty, elbow=epositive, wrist=wpositive, fatherId=fReference[0]}
  [271] = {x=-654.167, y=221.247, rx=180, rz=159.988, shoulder=lefty, elbow=epositive, wrist=wpositive, fatherId=fReference[0]}
  [272] = {x=-652.797, y=221.746, rx=180, rz=160.14, shoulder=lefty, elbow=epositive, wrist=wpositive, fatherId=fReference[0]}
  [273] = {x=-651.426, y=222.241, rx=180, rz=160.293, shoulder=lefty, elbow=epositive, wrist=wpositive, fatherId=fReference[0]}
  [274] = {x=-650.055, y=222.732, rx=180, rz=160.446, shoulder=lefty, elbow=epositive, wrist=wpositive, fatherId=fReference[0]}
  [275] = {x=-648.683, y=223.219, rx=-180, rz=160.6, shoulder=lefty, elbow=epositive, wrist=wpositive, fatherId=fReference[0]}
  [276] = {x=-647.31, y=223.703, rx=180, rz=160.755, shoulder=lefty, elbow=epositive, wrist=wpositive, fatherId=fReference[0]}
  [277] = {x=-645.937, y=224.182, rx=180, rz=160.91, shoulder=lefty, elbow=epositive, wrist=wpositive, fatherId=fReference[0]}
  [278] = {x=-644.562, y=224.658, rx=180, rz=161.066, shoulder=lefty, elbow=epositive, wrist=wpositive, fatherId=fReference[0]}
  [279] = {x=-643.188, y=225.129, rx=180, rz=161.223, shoulder=lefty, elbow=epositive, wrist=wpositive, fatherId=fReference[0]}
  [280] = {x=-641.812, y=225.597, rx=180, rz=161.381, shoulder=lefty, elbow=epositive, wrist=wpositive, fatherId=fReference[0]}
  [281] = {x=-640.436, y=226.061, rx=180, rz=161.539, shoulder=lefty, elbow=epositive, wrist=wpositive, fatherId=fReference[0]}
  [282] = {x=-639.06, y=226.52, rx=180, rz=161.698, shoulder=lefty, elbow=epositive, wrist=wpositive, fatherId=fReference[0]}
  [283] = {x=-637.682, y=226.976, rx=180, rz=161.857, shoulder=lefty, elbow=epositive, wrist=wpositive, fatherId=fReference[0]}
  [284] = {x=-636.304, y=227.427, rx=-180, rz=162.017, shoulder=lefty, elbow=epositive, wrist=wpositive, fatherId=fReference[0]}
  [285] = {x=-634.925, y=227.875, rx=180, rz=162.178, shoulder=lefty, elbow=epositive, wrist=wpositive, fatherId=fReference[0]}
  [286] = {x=-633.546, y=228.318, rx=-180, rz=162.34, shoulder=lefty, elbow=epositive, wrist=wpositive, fatherId=fReference[0]}
  [287] = {x=-632.166, y=228.758, rx=180, rz=162.502, shoulder=lefty, elbow=epositive, wrist=wpositive, fatherId=fReference[0]}
  [288] = {x=-630.786, y=229.193, rx=180, rz=162.665, shoulder=lefty, elbow=epositive, wrist=wpositive, fatherId=fReference[0]}
  [289] = {x=-629.404, y=229.624, rx=180, rz=162.829, shoulder=lefty, elbow=epositive, wrist=wpositive, fatherId=fReference[0]}
  [290] = {x=-628.022, y=230.051, rx=180, rz=162.993, shoulder=lefty, elbow=epositive, wrist=wpositive, fatherId=fReference[0]}
  [291] = {x=-626.64, y=230.474, rx=180, rz=163.158, shoulder=lefty, elbow=epositive, wrist=wpositive, fatherId=fReference[0]}
  [292] = {x=-625.257, y=230.893, rx=-180, rz=163.324, shoulder=lefty, elbow=epositive, wrist=wpositive, fatherId=fReference[0]}
  [293] = {x=-623.873, y=231.307, rx=180, rz=163.49, shoulder=lefty, elbow=epositive, wrist=wpositive, fatherId=fReference[0]}
  [294] = {x=-622.489, y=231.717, rx=-180, rz=163.657, shoulder=lefty, elbow=epositive, wrist=wpositive, fatherId=fReference[0]}
  [295] = {x=-621.104, y=232.124, rx=-180, rz=163.824, shoulder=lefty, elbow=epositive, wrist=wpositive, fatherId=fReference[0]}
  [296] = {x=-619.718, y=232.526, rx=180, rz=163.993, shoulder=lefty, elbow=epositive, wrist=wpositive, fatherId=fReference[0]}
  [297] = {x=-618.332, y=232.923, rx=180, rz=164.161, shoulder=lefty, elbow=epositive, wrist=wpositive, fatherId=fReference[0]}
  [298] = {x=-616.945, y=233.317, rx=180, rz=164.331, shoulder=lefty, elbow=epositive, wrist=wpositive, fatherId=fReference[0]}
  [299] = {x=-615.558, y=233.706, rx=-180, rz=164.501, shoulder=lefty, elbow=epositive, wrist=wpositive, fatherId=fReference[0]}
  [300] = {x=-614.17, y=234.091, rx=180, rz=164.672, shoulder=lefty, elbow=epositive, wrist=wpositive, fatherId=fReference[0]}
  [301] = {x=-612.781, y=234.471, rx=180, rz=164.843, shoulder=lefty, elbow=epositive, wrist=wpositive, fatherId=fReference[0]}
  [302] = {x=-611.392, y=234.848, rx=180, rz=165.015, shoulder=lefty, elbow=epositive, wrist=wpositive, fatherId=fReference[0]}
  [303] = {x=-610.002, y=235.22, rx=180, rz=165.188, shoulder=lefty, elbow=epositive, wrist=wpositive, fatherId=fReference[0]}
  [304] = {x=-608.612, y=235.587, rx=180, rz=165.361, shoulder=lefty, elbow=epositive, wrist=wpositive, fatherId=fReference[0]}
  [305] = {x=-607.221, y=235.951, rx=-180, rz=165.535, shoulder=lefty, elbow=epositive, wrist=wpositive, fatherId=fReference[0]}
  [306] = {x=-605.829, y=236.31, rx=-180, rz=165.71, shoulder=lefty, elbow=epositive, wrist=wpositive, fatherId=fReference[0]}
  [307] = {x=-604.437, y=236.664, rx=180, rz=165.885, shoulder=lefty, elbow=epositive, wrist=wpositive, fatherId=fReference[0]}
  [308] = {x=-603.045, y=237.014, rx=-180, rz=166.061, shoulder=lefty, elbow=epositive, wrist=wpositive, fatherId=fReference[0]}
  [309] = {x=-601.652, y=237.36, rx=180, rz=166.237, shoulder=lefty, elbow=epositive, wrist=wpositive, fatherId=fReference[0]}
  [310] = {x=-600.258, y=237.701, rx=-180, rz=166.414, shoulder=lefty, elbow=epositive, wrist=wpositive, fatherId=fReference[0]}
  [311] = {x=-598.864, y=238.038, rx=180, rz=166.591, shoulder=lefty, elbow=epositive, wrist=wpositive, fatherId=fReference[0]}
  [312] = {x=-597.469, y=238.371, rx=180, rz=166.77, shoulder=lefty, elbow=epositive, wrist=wpositive, fatherId=fReference[0]}
  [313] = {x=-596.074, y=238.699, rx=180, rz=166.948, shoulder=lefty, elbow=epositive, wrist=wpositive, fatherId=fReference[0]}
  [314] = {x=-594.678, y=239.023, rx=180, rz=167.127, shoulder=lefty, elbow=epositive, wrist=wpositive, fatherId=fReference[0]}
  [315] = {x=-593.281, y=239.342, rx=180, rz=167.307, shoulder=lefty, elbow=epositive, wrist=wpositive, fatherId=fReference[0]}
  [316] = {x=-591.885, y=239.656, rx=-180, rz=167.487, shoulder=lefty, elbow=epositive, wrist=wpositive, fatherId=fReference[0]}
  [317] = {x=-590.487, y=239.966, rx=180, rz=167.668, shoulder=lefty, elbow=epositive, wrist=wpositive, fatherId=fReference[0]}
  [318] = {x=-589.09, y=240.272, rx=180, rz=167.85, shoulder=lefty, elbow=epositive, wrist=wpositive, fatherId=fReference[0]}
  [319] = {x=-587.691, y=240.573, rx=180, rz=168.032, shoulder=lefty, elbow=epositive, wrist=wpositive, fatherId=fReference[0]}
  [320] = {x=-586.292, y=240.869, rx=180, rz=168.214, shoulder=lefty, elbow=epositive, wrist=wpositive, fatherId=fReference[0]}
  [321] = {x=-584.893, y=241.161, rx=180, rz=168.397, shoulder=lefty, elbow=epositive, wrist=wpositive, fatherId=fReference[0]}
  [322] = {x=-583.493, y=241.449, rx=180, rz=168.581, shoulder=lefty, elbow=epositive, wrist=wpositive, fatherId=fReference[0]}
  [323] = {x=-582.093, y=241.732, rx=180, rz=168.765, shoulder=lefty, elbow=epositive, wrist=wpositive, fatherId=fReference[0]}
  [324] = {x=-580.693, y=242.01, rx=180, rz=168.949, shoulder=lefty, elbow=epositive, wrist=wpositive, fatherId=fReference[0]}
  [325] = {x=-579.292, y=242.283, rx=-180, rz=169.134, shoulder=lefty, elbow=epositive, wrist=wpositive, fatherId=fReference[0]}
  [326] = {x=-577.89, y=242.553, rx=180, rz=169.32, shoulder=lefty, elbow=epositive, wrist=wpositive, fatherId=fReference[0]}
  [327] = {x=-576.488, y=242.817, rx=180, rz=169.506, shoulder=lefty, elbow=epositive, wrist=wpositive, fatherId=fReference[0]}
  [328] = {x=-575.086, y=243.077, rx=-180, rz=169.692, shoulder=lefty, elbow=epositive, wrist=wpositive, fatherId=fReference[0]}
  [329] = {x=-573.683, y=243.332, rx=-180, rz=169.879, shoulder=lefty, elbow=epositive, wrist=wpositive, fatherId=fReference[0]}
  [330] = {x=-572.279, y=243.582, rx=180, rz=170.067, shoulder=lefty, elbow=epositive, wrist=wpositive, fatherId=fReference[0]}
  [331] = {x=-570.876, y=243.828, rx=-180, rz=170.255, shoulder=lefty, elbow=epositive, wrist=wpositive, fatherId=fReference[0]}
  [332] = {x=-569.472, y=244.069, rx=-180, rz=170.443, shoulder=lefty, elbow=epositive, wrist=wpositive, fatherId=fReference[0]}
  [333] = {x=-568.067, y=244.306, rx=180, rz=170.632, shoulder=lefty, elbow=epositive, wrist=wpositive, fatherId=fReference[0]}
  [334] = {x=-566.662, y=244.538, rx=180, rz=170.821, shoulder=lefty, elbow=epositive, wrist=wpositive, fatherId=fReference[0]}
  [335] = {x=-565.257, y=244.765, rx=180, rz=171.011, shoulder=lefty, elbow=epositive, wrist=wpositive, fatherId=fReference[0]}
  [336] = {x=-563.852, y=244.987, rx=-180, rz=171.201, shoulder=lefty, elbow=epositive, wrist=wpositive, fatherId=fReference[0]}
  [337] = {x=-562.446, y=245.205, rx=-180, rz=171.391, shoulder=lefty, elbow=epositive, wrist=wpositive, fatherId=fReference[0]}
  [338] = {x=-561.039, y=245.417, rx=180, rz=171.582, shoulder=lefty, elbow=epositive, wrist=wpositive, fatherId=fReference[0]}
  [339] = {x=-559.632, y=245.626, rx=180, rz=171.774, shoulder=lefty, elbow=epositive, wrist=wpositive, fatherId=fReference[0]}
  [340] = {x=-558.225, y=245.829, rx=180, rz=171.965, shoulder=lefty, elbow=epositive, wrist=wpositive, fatherId=fReference[0]}
  [341] = {x=-556.818, y=246.028, rx=180, rz=172.157, shoulder=lefty, elbow=epositive, wrist=wpositive, fatherId=fReference[0]}
  [342] = {x=-555.41, y=246.222, rx=180, rz=172.35, shoulder=lefty, elbow=epositive, wrist=wpositive, fatherId=fReference[0]}
  [343] = {x=-554.002, y=246.411, rx=180, rz=172.543, shoulder=lefty, elbow=epositive, wrist=wpositive, fatherId=fReference[0]}
  [344] = {x=-552.594, y=246.595, rx=-180, rz=172.736, shoulder=lefty, elbow=epositive, wrist=wpositive, fatherId=fReference[0]}
  [345] = {x=-551.185, y=246.775, rx=180, rz=172.929, shoulder=lefty, elbow=epositive, wrist=wpositive, fatherId=fReference[0]}
  [346] = {x=-549.776, y=246.949, rx=180, rz=173.123, shoulder=lefty, elbow=epositive, wrist=wpositive, fatherId=fReference[0]}
  [347] = {x=-548.367, y=247.119, rx=180, rz=173.317, shoulder=lefty, elbow=epositive, wrist=wpositive, fatherId=fReference[0]}
  [348] = {x=-546.957, y=247.285, rx=-180, rz=173.512, shoulder=lefty, elbow=epositive, wrist=wpositive, fatherId=fReference[0]}
  [349] = {x=-545.548, y=247.445, rx=180, rz=173.707, shoulder=lefty, elbow=epositive, wrist=wpositive, fatherId=fReference[0]}
  [350] = {x=-544.137, y=247.6, rx=180, rz=173.902, shoulder=lefty, elbow=epositive, wrist=wpositive, fatherId=fReference[0]}
  [351] = {x=-542.727, y=247.751, rx=180, rz=174.097, shoulder=lefty, elbow=epositive, wrist=wpositive, fatherId=fReference[0]}
  [352] = {x=-541.316, y=247.897, rx=180, rz=174.293, shoulder=lefty, elbow=epositive, wrist=wpositive, fatherId=fReference[0]}
  [353] = {x=-539.905, y=248.038, rx=180, rz=174.489, shoulder=lefty, elbow=epositive, wrist=wpositive, fatherId=fReference[0]}
  [354] = {x=-538.494, y=248.174, rx=-180, rz=174.685, shoulder=lefty, elbow=epositive, wrist=wpositive, fatherId=fReference[0]}
  [355] = {x=-537.083, y=248.305, rx=180, rz=174.882, shoulder=lefty, elbow=epositive, wrist=wpositive, fatherId=fReference[0]}
  [356] = {x=-535.671, y=248.432, rx=180, rz=175.079, shoulder=lefty, elbow=epositive, wrist=wpositive, fatherId=fReference[0]}
  [357] = {x=-534.26, y=248.553, rx=180, rz=175.276, shoulder=lefty, elbow=epositive, wrist=wpositive, fatherId=fReference[0]}
  [358] = {x=-532.848, y=248.67, rx=-180, rz=175.473, shoulder=lefty, elbow=epositive, wrist=wpositive, fatherId=fReference[0]}
  [359] = {x=-531.435, y=248.782, rx=180, rz=175.671, shoulder=lefty, elbow=epositive, wrist=wpositive, fatherId=fReference[0]}
  [360] = {x=-530.023, y=248.889, rx=180, rz=175.868, shoulder=lefty, elbow=epositive, wrist=wpositive, fatherId=fReference[0]}
  [361] = {x=-528.61, y=248.991, rx=-180, rz=176.066, shoulder=lefty, elbow=epositive, wrist=wpositive, fatherId=fReference[0]}
  [362] = {x=-527.198, y=249.088, rx=-180, rz=176.264, shoulder=lefty, elbow=epositive, wrist=wpositive, fatherId=fReference[0]}
  [363] = {x=-525.785, y=249.18, rx=180, rz=176.463, shoulder=lefty, elbow=epositive, wrist=wpositive, fatherId=fReference[0]}
  [364] = {x=-524.372, y=249.268, rx=-180, rz=176.661, shoulder=lefty, elbow=epositive, wrist=wpositive, fatherId=fReference[0]}
  [365] = {x=-522.958, y=249.35, rx=180, rz=176.86, shoulder=lefty, elbow=epositive, wrist=wpositive, fatherId=fReference[0]}
  [366] = {x=-521.545, y=249.428, rx=180, rz=177.059, shoulder=lefty, elbow=epositive, wrist=wpositive, fatherId=fReference[0]}
  [367] = {x=-520.132, y=249.5, rx=180, rz=177.258, shoulder=lefty, elbow=epositive, wrist=wpositive, fatherId=fReference[0]}
  [368] = {x=-518.718, y=249.568, rx=-180, rz=177.457, shoulder=lefty, elbow=epositive, wrist=wpositive, fatherId=fReference[0]}
  [369] = {x=-517.304, y=249.631, rx=180, rz=177.656, shoulder=lefty, elbow=epositive, wrist=wpositive, fatherId=fReference[0]}
  [370] = {x=-515.89, y=249.689, rx=180, rz=177.855, shoulder=lefty, elbow=epositive, wrist=wpositive, fatherId=fReference[0]}
  [371] = {x=-514.476, y=249.742, rx=180, rz=178.055, shoulder=lefty, elbow=epositive, wrist=wpositive, fatherId=fReference[0]}
  [372] = {x=-513.062, y=249.79, rx=180, rz=178.254, shoulder=lefty, elbow=epositive, wrist=wpositive, fatherId=fReference[0]}
  [373] = {x=-511.648, y=249.833, rx=-180, rz=178.454, shoulder=lefty, elbow=epositive, wrist=wpositive, fatherId=fReference[0]}
  [374] = {x=-510.234, y=249.871, rx=180, rz=178.654, shoulder=lefty, elbow=epositive, wrist=wpositive, fatherId=fReference[0]}
  [375] = {x=-508.82, y=249.904, rx=180, rz=178.853, shoulder=lefty, elbow=epositive, wrist=wpositive, fatherId=fReference[0]}
  [376] = {x=-507.405, y=249.932, rx=-180, rz=179.053, shoulder=lefty, elbow=epositive, wrist=wpositive, fatherId=fReference[0]}
  [377] = {x=-505.991, y=249.956, rx=-180, rz=179.253, shoulder=lefty, elbow=epositive, wrist=wpositive, fatherId=fReference[0]}
  [378] = {x=-504.577, y=249.974, rx=-180, rz=179.453, shoulder=lefty, elbow=epositive, wrist=wpositive, fatherId=fReference[0]}
  [379] = {x=-503.162, y=249.988, rx=-180, rz=179.653, shoulder=lefty, elbow=epositive, wrist=wpositive, fatherId=fReference[0]}
  [380] = {x=-501.748, y=249.996, rx=180, rz=179.853, shoulder=lefty, elbow=epositive, wrist=wpositive, fatherId=fReference[0]}
  [381] = {x=-500.333, y=250, rx=-180, rz=-179.947, shoulder=lefty, elbow=epositive, wrist=wpositive, fatherId=fReference[0]}
  [382] = {x=-498.919, y=249.999, rx=180, rz=-179.747, shoulder=lefty, elbow=epositive, wrist=wpositive, fatherId=fReference[0]}
  [383] = {x=-497.504, y=249.992, rx=180, rz=-179.547, shoulder=lefty, elbow=epositive, wrist=wpositive, fatherId=fReference[0]}
  [384] = {x=-496.09, y=249.981, rx=180, rz=-179.347, shoulder=lefty, elbow=epositive, wrist=wpositive, fatherId=fReference[0]}
  [385] = {x=-494.676, y=249.965, rx=-180, rz=-179.147, shoulder=lefty, elbow=epositive, wrist=wpositive, fatherId=fReference[0]}
  [386] = {x=-493.261, y=249.944, rx=180, rz=-178.947, shoulder=lefty, elbow=epositive, wrist=wpositive, fatherId=fReference[0]}
  [387] = {x=-491.847, y=249.918, rx=180, rz=-178.748, shoulder=lefty, elbow=epositive, wrist=wpositive, fatherId=fReference[0]}
  [388] = {x=-490.433, y=249.887, rx=-180, rz=-178.548, shoulder=lefty, elbow=epositive, wrist=wpositive, fatherId=fReference[0]}
  [389] = {x=-489.019, y=249.851, rx=-180, rz=-178.348, shoulder=lefty, elbow=epositive, wrist=wpositive, fatherId=fReference[0]}
  [390] = {x=-487.604, y=249.81, rx=-180, rz=-178.149, shoulder=lefty, elbow=epositive, wrist=wpositive, fatherId=fReference[0]}
  [391] = {x=-486.19, y=249.765, rx=180, rz=-177.949, shoulder=lefty, elbow=epositive, wrist=wpositive, fatherId=fReference[0]}
  [392] = {x=-484.776, y=249.714, rx=180, rz=-177.75, shoulder=lefty, elbow=epositive, wrist=wpositive, fatherId=fReference[0]}
  [393] = {x=-483.363, y=249.659, rx=180, rz=-177.551, shoulder=lefty, elbow=epositive, wrist=wpositive, fatherId=fReference[0]}
  [394] = {x=-481.949, y=249.598, rx=-180, rz=-177.351, shoulder=lefty, elbow=epositive, wrist=wpositive, fatherId=fReference[0]}
  [395] = {x=-480.535, y=249.533, rx=-180, rz=-177.152, shoulder=lefty, elbow=epositive, wrist=wpositive, fatherId=fReference[0]}
  [396] = {x=-479.122, y=249.462, rx=180, rz=-176.954, shoulder=lefty, elbow=epositive, wrist=wpositive, fatherId=fReference[0]}
  [397] = {x=-477.708, y=249.387, rx=180, rz=-176.755, shoulder=lefty, elbow=epositive, wrist=wpositive, fatherId=fReference[0]}
  [398] = {x=-476.295, y=249.307, rx=180, rz=-176.556, shoulder=lefty, elbow=epositive, wrist=wpositive, fatherId=fReference[0]}
  [399] = {x=-474.882, y=249.222, rx=180, rz=-176.358, shoulder=lefty, elbow=epositive, wrist=wpositive, fatherId=fReference[0]}
  [400] = {x=-473.469, y=249.132, rx=-180, rz=-176.16, shoulder=lefty, elbow=epositive, wrist=wpositive, fatherId=fReference[0]}
  [401] = {x=-472.056, y=249.037, rx=180, rz=-175.962, shoulder=lefty, elbow=epositive, wrist=wpositive, fatherId=fReference[0]}
  [402] = {x=-470.643, y=248.937, rx=-180, rz=-175.764, shoulder=lefty, elbow=epositive, wrist=wpositive, fatherId=fReference[0]}
  [403] = {x=-469.231, y=248.833, rx=180, rz=-175.566, shoulder=lefty, elbow=epositive, wrist=wpositive, fatherId=fReference[0]}
  [404] = {x=-467.819, y=248.723, rx=-180, rz=-175.369, shoulder=lefty, elbow=epositive, wrist=wpositive, fatherId=fReference[0]}
  [405] = {x=-466.407, y=248.609, rx=180, rz=-175.172, shoulder=lefty, elbow=epositive, wrist=wpositive, fatherId=fReference[0]}
  [406] = {x=-464.995, y=248.49, rx=180, rz=-174.975, shoulder=lefty, elbow=epositive, wrist=wpositive, fatherId=fReference[0]}
  [407] = {x=-463.583, y=248.366, rx=-180, rz=-174.778, shoulder=lefty, elbow=epositive, wrist=wpositive, fatherId=fReference[0]}
  [408] = {x=-462.172, y=248.237, rx=180, rz=-174.582, shoulder=lefty, elbow=epositive, wrist=wpositive, fatherId=fReference[0]}
  [409] = {x=-460.76, y=248.103, rx=180, rz=-174.386, shoulder=lefty, elbow=epositive, wrist=wpositive, fatherId=fReference[0]}
  [410] = {x=-459.349, y=247.964, rx=-180, rz=-174.19, shoulder=lefty, elbow=epositive, wrist=wpositive, fatherId=fReference[0]}
  [411] = {x=-457.939, y=247.82, rx=180, rz=-173.994, shoulder=lefty, elbow=epositive, wrist=wpositive, fatherId=fReference[0]}
  [412] = {x=-456.528, y=247.672, rx=-180, rz=-173.799, shoulder=lefty, elbow=epositive, wrist=wpositive, fatherId=fReference[0]}
  [413] = {x=-455.118, y=247.519, rx=180, rz=-173.604, shoulder=lefty, elbow=epositive, wrist=wpositive, fatherId=fReference[0]}
  [414] = {x=-453.708, y=247.361, rx=180, rz=-173.409, shoulder=lefty, elbow=epositive, wrist=wpositive, fatherId=fReference[0]}
  [415] = {x=-452.298, y=247.198, rx=180, rz=-173.215, shoulder=lefty, elbow=epositive, wrist=wpositive, fatherId=fReference[0]}
  [416] = {x=-450.889, y=247.03, rx=180, rz=-173.021, shoulder=lefty, elbow=epositive, wrist=wpositive, fatherId=fReference[0]}
  [417] = {x=-449.48, y=246.858, rx=-180, rz=-172.827, shoulder=lefty, elbow=epositive, wrist=wpositive, fatherId=fReference[0]}
  [418] = {x=-448.071, y=246.68, rx=180, rz=-172.634, shoulder=lefty, elbow=epositive, wrist=wpositive, fatherId=fReference[0]}
  [419] = {x=-446.663, y=246.498, rx=180, rz=-172.441, shoulder=lefty, elbow=epositive, wrist=wpositive, fatherId=fReference[0]}
  [420] = {x=-445.254, y=246.312, rx=180, rz=-172.248, shoulder=lefty, elbow=epositive, wrist=wpositive, fatherId=fReference[0]}
  [421] = {x=-443.847, y=246.12, rx=180, rz=-172.056, shoulder=lefty, elbow=epositive, wrist=wpositive, fatherId=fReference[0]}
  [422] = {x=-442.439, y=245.923, rx=-180, rz=-171.864, shoulder=lefty, elbow=epositive, wrist=wpositive, fatherId=fReference[0]}
  [423] = {x=-441.032, y=245.722, rx=-180, rz=-171.673, shoulder=lefty, elbow=epositive, wrist=wpositive, fatherId=fReference[0]}
  [424] = {x=-439.625, y=245.516, rx=-180, rz=-171.482, shoulder=lefty, elbow=epositive, wrist=wpositive, fatherId=fReference[0]}
  [425] = {x=-438.218, y=245.306, rx=-180, rz=-171.291, shoulder=lefty, elbow=epositive, wrist=wpositive, fatherId=fReference[0]}
  [426] = {x=-436.812, y=245.09, rx=-180, rz=-171.101, shoulder=lefty, elbow=epositive, wrist=wpositive, fatherId=fReference[0]}
  [427] = {x=-435.406, y=244.87, rx=180, rz=-170.911, shoulder=lefty, elbow=epositive, wrist=wpositive, fatherId=fReference[0]}
  [428] = {x=-434.001, y=244.645, rx=180, rz=-170.721, shoulder=lefty, elbow=epositive, wrist=wpositive, fatherId=fReference[0]}
  [429] = {x=-432.596, y=244.416, rx=180, rz=-170.532, shoulder=lefty, elbow=epositive, wrist=wpositive, fatherId=fReference[0]}
  [430] = {x=-431.191, y=244.182, rx=-180, rz=-170.344, shoulder=lefty, elbow=epositive, wrist=wpositive, fatherId=fReference[0]}
  [431] = {x=-429.787, y=243.943, rx=180, rz=-170.156, shoulder=lefty, elbow=epositive, wrist=wpositive, fatherId=fReference[0]}
  [432] = {x=-428.383, y=243.699, rx=-180, rz=-169.968, shoulder=lefty, elbow=epositive, wrist=wpositive, fatherId=fReference[0]}
  [433] = {x=-426.98, y=243.451, rx=180, rz=-169.781, shoulder=lefty, elbow=epositive, wrist=wpositive, fatherId=fReference[0]}
  [434] = {x=-425.577, y=243.198, rx=180, rz=-169.594, shoulder=lefty, elbow=epositive, wrist=wpositive, fatherId=fReference[0]}
  [435] = {x=-424.174, y=242.94, rx=-180, rz=-169.408, shoulder=lefty, elbow=epositive, wrist=wpositive, fatherId=fReference[0]}
  [436] = {x=-422.772, y=242.678, rx=180, rz=-169.222, shoulder=lefty, elbow=epositive, wrist=wpositive, fatherId=fReference[0]}
  [437] = {x=-421.37, y=242.411, rx=180, rz=-169.037, shoulder=lefty, elbow=epositive, wrist=wpositive, fatherId=fReference[0]}
  [438] = {x=-419.969, y=242.14, rx=-180, rz=-168.852, shoulder=lefty, elbow=epositive, wrist=wpositive, fatherId=fReference[0]}
  [439] = {x=-418.568, y=241.864, rx=-180, rz=-168.667, shoulder=lefty, elbow=epositive, wrist=wpositive, fatherId=fReference[0]}
  [440] = {x=-417.167, y=241.583, rx=-180, rz=-168.484, shoulder=lefty, elbow=epositive, wrist=wpositive, fatherId=fReference[0]}
  [441] = {x=-415.767, y=241.298, rx=-180, rz=-168.3, shoulder=lefty, elbow=epositive, wrist=wpositive, fatherId=fReference[0]}
  [442] = {x=-414.368, y=241.008, rx=180, rz=-168.118, shoulder=lefty, elbow=epositive, wrist=wpositive, fatherId=fReference[0]}
  [443] = {x=-412.969, y=240.713, rx=180, rz=-167.935, shoulder=lefty, elbow=epositive, wrist=wpositive, fatherId=fReference[0]}
  [444] = {x=-411.57, y=240.415, rx=180, rz=-167.754, shoulder=lefty, elbow=epositive, wrist=wpositive, fatherId=fReference[0]}
  [445] = {x=-410.172, y=240.111, rx=-180, rz=-167.573, shoulder=lefty, elbow=epositive, wrist=wpositive, fatherId=fReference[0]}
  [446] = {x=-408.775, y=239.803, rx=-180, rz=-167.392, shoulder=lefty, elbow=epositive, wrist=wpositive, fatherId=fReference[0]}
  [447] = {x=-407.378, y=239.491, rx=-180, rz=-167.212, shoulder=lefty, elbow=epositive, wrist=wpositive, fatherId=fReference[0]}
  [448] = {x=-405.981, y=239.174, rx=180, rz=-167.033, shoulder=lefty, elbow=epositive, wrist=wpositive, fatherId=fReference[0]}
  [449] = {x=-404.585, y=238.852, rx=-180, rz=-166.854, shoulder=lefty, elbow=epositive, wrist=wpositive, fatherId=fReference[0]}
  [450] = {x=-403.189, y=238.526, rx=180, rz=-166.675, shoulder=lefty, elbow=epositive, wrist=wpositive, fatherId=fReference[0]}
  [451] = {x=-401.794, y=238.196, rx=-180, rz=-166.498, shoulder=lefty, elbow=epositive, wrist=wpositive, fatherId=fReference[0]}
  [452] = {x=-400.4, y=237.861, rx=180, rz=-166.32, shoulder=lefty, elbow=epositive, wrist=wpositive, fatherId=fReference[0]}
  [453] = {x=-399.006, y=237.522, rx=-180, rz=-166.144, shoulder=lefty, elbow=epositive, wrist=wpositive, fatherId=fReference[0]}
  [454] = {x=-397.613, y=237.178, rx=-180, rz=-165.968, shoulder=lefty, elbow=epositive, wrist=wpositive, fatherId=fReference[0]}
  [455] = {x=-396.22, y=236.83, rx=-180, rz=-165.792, shoulder=lefty, elbow=epositive, wrist=wpositive, fatherId=fReference[0]}
  [456] = {x=-394.827, y=236.477, rx=180, rz=-165.618, shoulder=lefty, elbow=epositive, wrist=wpositive, fatherId=fReference[0]}
  [457] = {x=-393.436, y=236.12, rx=180, rz=-165.443, shoulder=lefty, elbow=epositive, wrist=wpositive, fatherId=fReference[0]}
  [458] = {x=-392.044, y=235.759, rx=180, rz=-165.27, shoulder=lefty, elbow=epositive, wrist=wpositive, fatherId=fReference[0]}
  [459] = {x=-390.654, y=235.394, rx=-180, rz=-165.097, shoulder=lefty, elbow=epositive, wrist=wpositive, fatherId=fReference[0]}
  [460] = {x=-389.264, y=235.024, rx=-180, rz=-164.924, shoulder=lefty, elbow=epositive, wrist=wpositive, fatherId=fReference[0]}
  [461] = {x=-387.874, y=234.649, rx=180, rz=-164.753, shoulder=lefty, elbow=epositive, wrist=wpositive, fatherId=fReference[0]}
  [462] = {x=-386.485, y=234.271, rx=180, rz=-164.582, shoulder=lefty, elbow=epositive, wrist=wpositive, fatherId=fReference[0]}
  [463] = {x=-385.097, y=233.888, rx=180, rz=-164.411, shoulder=lefty, elbow=epositive, wrist=wpositive, fatherId=fReference[0]}
  [464] = {x=-383.709, y=233.501, rx=-180, rz=-164.241, shoulder=lefty, elbow=epositive, wrist=wpositive, fatherId=fReference[0]}
  [465] = {x=-382.322, y=233.109, rx=-180, rz=-164.072, shoulder=lefty, elbow=epositive, wrist=wpositive, fatherId=fReference[0]}
  [466] = {x=-380.936, y=232.714, rx=-180, rz=-163.904, shoulder=lefty, elbow=epositive, wrist=wpositive, fatherId=fReference[0]}
  [467] = {x=-379.55, y=232.314, rx=-180, rz=-163.736, shoulder=lefty, elbow=epositive, wrist=wpositive, fatherId=fReference[0]}
  [468] = {x=-378.164, y=231.909, rx=-180, rz=-163.568, shoulder=lefty, elbow=epositive, wrist=wpositive, fatherId=fReference[0]}
  [469] = {x=-376.78, y=231.501, rx=-180, rz=-163.402, shoulder=lefty, elbow=epositive, wrist=wpositive, fatherId=fReference[0]}
  [470] = {x=-375.395, y=231.089, rx=180, rz=-163.236, shoulder=lefty, elbow=epositive, wrist=wpositive, fatherId=fReference[0]}
  [471] = {x=-374.012, y=230.672, rx=180, rz=-163.071, shoulder=lefty, elbow=epositive, wrist=wpositive, fatherId=fReference[0]}
  [472] = {x=-372.629, y=230.251, rx=-180, rz=-162.906, shoulder=lefty, elbow=epositive, wrist=wpositive, fatherId=fReference[0]}
  [473] = {x=-371.247, y=229.826, rx=-180, rz=-162.742, shoulder=lefty, elbow=epositive, wrist=wpositive, fatherId=fReference[0]}
  [474] = {x=-369.865, y=229.397, rx=-180, rz=-162.579, shoulder=lefty, elbow=epositive, wrist=wpositive, fatherId=fReference[0]}
  [475] = {x=-368.484, y=228.963, rx=180, rz=-162.416, shoulder=lefty, elbow=epositive, wrist=wpositive, fatherId=fReference[0]}
  [476] = {x=-367.104, y=228.526, rx=-180, rz=-162.254, shoulder=lefty, elbow=epositive, wrist=wpositive, fatherId=fReference[0]}
  [477] = {x=-365.724, y=228.084, rx=-180, rz=-162.093, shoulder=lefty, elbow=epositive, wrist=wpositive, fatherId=fReference[0]}
  [478] = {x=-364.345, y=227.639, rx=180, rz=-161.932, shoulder=lefty, elbow=epositive, wrist=wpositive, fatherId=fReference[0]}
  [479] = {x=-362.966, y=227.189, rx=180, rz=-161.772, shoulder=lefty, elbow=epositive, wrist=wpositive, fatherId=fReference[0]}
  [480] = {x=-361.588, y=226.735, rx=-180, rz=-161.613, shoulder=lefty, elbow=epositive, wrist=wpositive, fatherId=fReference[0]}
  [481] = {x=-360.211, y=226.277, rx=180, rz=-161.455, shoulder=lefty, elbow=epositive, wrist=wpositive, fatherId=fReference[0]}
  [482] = {x=-358.835, y=225.816, rx=180, rz=-161.297, shoulder=lefty, elbow=epositive, wrist=wpositive, fatherId=fReference[0]}
  [483] = {x=-357.459, y=225.35, rx=180, rz=-161.14, shoulder=lefty, elbow=epositive, wrist=wpositive, fatherId=fReference[0]}
  [484] = {x=-356.084, y=224.88, rx=-180, rz=-160.983, shoulder=lefty, elbow=epositive, wrist=wpositive, fatherId=fReference[0]}
  [485] = {x=-354.709, y=224.406, rx=180, rz=-160.828, shoulder=lefty, elbow=epositive, wrist=wpositive, fatherId=fReference[0]}
  [486] = {x=-353.335, y=223.929, rx=-180, rz=-160.673, shoulder=lefty, elbow=epositive, wrist=wpositive, fatherId=fReference[0]}
  [487] = {x=-351.962, y=223.447, rx=-180, rz=-160.518, shoulder=lefty, elbow=epositive, wrist=wpositive, fatherId=fReference[0]}
  [488] = {x=-350.59, y=222.961, rx=180, rz=-160.365, shoulder=lefty, elbow=epositive, wrist=wpositive, fatherId=fReference[0]}
  [489] = {x=-349.218, y=222.472, rx=-180, rz=-160.212, shoulder=lefty, elbow=epositive, wrist=wpositive, fatherId=fReference[0]}
  [490] = {x=-347.847, y=221.979, rx=180, rz=-160.06, shoulder=lefty, elbow=epositive, wrist=wpositive, fatherId=fReference[0]}
  [491] = {x=-346.476, y=221.482, rx=-180, rz=-159.908, shoulder=lefty, elbow=epositive, wrist=wpositive, fatherId=fReference[0]}
  [492] = {x=-345.107, y=220.98, rx=-180, rz=-159.757, shoulder=lefty, elbow=epositive, wrist=wpositive, fatherId=fReference[0]}
  [493] = {x=-343.737, y=220.476, rx=180, rz=-159.607, shoulder=lefty, elbow=epositive, wrist=wpositive, fatherId=fReference[0]}
  [494] = {x=-342.369, y=219.967, rx=180, rz=-159.458, shoulder=lefty, elbow=epositive, wrist=wpositive, fatherId=fReference[0]}
  [495] = {x=-341.001, y=219.454, rx=180, rz=-159.309, shoulder=lefty, elbow=epositive, wrist=wpositive, fatherId=fReference[0]}
  [496] = {x=-339.634, y=218.938, rx=180, rz=-159.161, shoulder=lefty, elbow=epositive, wrist=wpositive, fatherId=fReference[0]}
  [497] = {x=-338.268, y=218.418, rx=180, rz=-159.014, shoulder=lefty, elbow=epositive, wrist=wpositive, fatherId=fReference[0]}
  [498] = {x=-336.903, y=217.894, rx=-180, rz=-158.868, shoulder=lefty, elbow=epositive, wrist=wpositive, fatherId=fReference[0]}
  [499] = {x=-335.538, y=217.367, rx=-180, rz=-158.722, shoulder=lefty, elbow=epositive, wrist=wpositive, fatherId=fReference[0]}
  [500] = {x=-334.173, y=216.835, rx=-180, rz=-158.577, shoulder=lefty, elbow=epositive, wrist=wpositive, fatherId=fReference[0]}
  [501] = {x=-332.81, y=216.3, rx=-180, rz=-158.433, shoulder=lefty, elbow=epositive, wrist=wpositive, fatherId=fReference[0]}
  [502] = {x=-331.447, y=215.762, rx=180, rz=-158.289, shoulder=lefty, elbow=epositive, wrist=wpositive, fatherId=fReference[0]}
  [503] = {x=-330.085, y=215.219, rx=180, rz=-158.146, shoulder=lefty, elbow=epositive, wrist=wpositive, fatherId=fReference[0]}
  [504] = {x=-328.724, y=214.674, rx=180, rz=-158.004, shoulder=lefty, elbow=epositive, wrist=wpositive, fatherId=fReference[0]}
  [505] = {x=-327.363, y=214.124, rx=-180, rz=-157.862, shoulder=lefty, elbow=epositive, wrist=wpositive, fatherId=fReference[0]}
  [506] = {x=-326.004, y=213.571, rx=180, rz=-157.722, shoulder=lefty, elbow=epositive, wrist=wpositive, fatherId=fReference[0]}
  [507] = {x=-324.644, y=213.014, rx=180, rz=-157.582, shoulder=lefty, elbow=epositive, wrist=wpositive, fatherId=fReference[0]}
  [508] = {x=-323.286, y=212.453, rx=-180, rz=-157.442, shoulder=lefty, elbow=epositive, wrist=wpositive, fatherId=fReference[0]}
  [509] = {x=-321.928, y=211.89, rx=-180, rz=-157.304, shoulder=lefty, elbow=epositive, wrist=wpositive, fatherId=fReference[0]}
  [510] = {x=-320.571, y=211.322, rx=180, rz=-157.166, shoulder=lefty, elbow=epositive, wrist=wpositive, fatherId=fReference[0]}
  [511] = {x=-319.215, y=210.751, rx=-180, rz=-157.029, shoulder=lefty, elbow=epositive, wrist=wpositive, fatherId=fReference[0]}
  [512] = {x=-317.86, y=210.176, rx=-180, rz=-156.893, shoulder=lefty, elbow=epositive, wrist=wpositive, fatherId=fReference[0]}
  [513] = {x=-316.505, y=209.598, rx=-180, rz=-156.757, shoulder=lefty, elbow=epositive, wrist=wpositive, fatherId=fReference[0]}
  [514] = {x=-315.151, y=209.017, rx=180, rz=-156.622, shoulder=lefty, elbow=epositive, wrist=wpositive, fatherId=fReference[0]}
  [515] = {x=-313.798, y=208.432, rx=180, rz=-156.488, shoulder=lefty, elbow=epositive, wrist=wpositive, fatherId=fReference[0]}
  [516] = {x=-312.445, y=207.843, rx=180, rz=-156.354, shoulder=lefty, elbow=epositive, wrist=wpositive, fatherId=fReference[0]}
  [517] = {x=-311.094, y=207.252, rx=-180, rz=-156.222, shoulder=lefty, elbow=epositive, wrist=wpositive, fatherId=fReference[0]}
  [518] = {x=-309.743, y=206.656, rx=180, rz=-156.09, shoulder=lefty, elbow=epositive, wrist=wpositive, fatherId=fReference[0]}
  [519] = {x=-308.392, y=206.058, rx=180, rz=-155.958, shoulder=lefty, elbow=epositive, wrist=wpositive, fatherId=fReference[0]}
  [520] = {x=-307.043, y=205.456, rx=180, rz=-155.828, shoulder=lefty, elbow=epositive, wrist=wpositive, fatherId=fReference[0]}
  [521] = {x=-305.694, y=204.85, rx=-180, rz=-155.698, shoulder=lefty, elbow=epositive, wrist=wpositive, fatherId=fReference[0]}
  [522] = {x=-304.346, y=204.242, rx=180, rz=-155.569, shoulder=lefty, elbow=epositive, wrist=wpositive, fatherId=fReference[0]}
  [523] = {x=-302.999, y=203.63, rx=-180, rz=-155.44, shoulder=lefty, elbow=epositive, wrist=wpositive, fatherId=fReference[0]}
  [524] = {x=-301.652, y=203.014, rx=-180, rz=-155.312, shoulder=lefty, elbow=epositive, wrist=wpositive, fatherId=fReference[0]}
  [525] = {x=-300.307, y=202.396, rx=-180, rz=-155.185, shoulder=lefty, elbow=epositive, wrist=wpositive, fatherId=fReference[0]}
  [526] = {x=-298.962, y=201.774, rx=-180, rz=-155.059, shoulder=lefty, elbow=epositive, wrist=wpositive, fatherId=fReference[0]}
  [527] = {x=-297.618, y=201.149, rx=180, rz=-154.934, shoulder=lefty, elbow=epositive, wrist=wpositive, fatherId=fReference[0]}
  [528] = {x=-296.274, y=200.52, rx=-180, rz=-154.809, shoulder=lefty, elbow=epositive, wrist=wpositive, fatherId=fReference[0]}
  [529] = {x=-294.931, y=199.889, rx=180, rz=-154.685, shoulder=lefty, elbow=epositive, wrist=wpositive, fatherId=fReference[0]}
  [530] = {x=-293.589, y=199.254, rx=-180, rz=-154.561, shoulder=lefty, elbow=epositive, wrist=wpositive, fatherId=fReference[0]}
  [531] = {x=-292.248, y=198.616, rx=-180, rz=-154.439, shoulder=lefty, elbow=epositive, wrist=wpositive, fatherId=fReference[0]}
  [532] = {x=-290.908, y=197.975, rx=180, rz=-154.317, shoulder=lefty, elbow=epositive, wrist=wpositive, fatherId=fReference[0]}
  [533] = {x=-289.568, y=197.331, rx=-180, rz=-154.195, shoulder=lefty, elbow=epositive, wrist=wpositive, fatherId=fReference[0]}
  [534] = {x=-288.229, y=196.683, rx=180, rz=-154.075, shoulder=lefty, elbow=epositive, wrist=wpositive, fatherId=fReference[0]}
  [535] = {x=-286.891, y=196.033, rx=180, rz=-153.955, shoulder=lefty, elbow=epositive, wrist=wpositive, fatherId=fReference[0]}
  [536] = {x=-285.554, y=195.379, rx=180, rz=-153.836, shoulder=lefty, elbow=epositive, wrist=wpositive, fatherId=fReference[0]}
  [537] = {x=-284.217, y=194.723, rx=180, rz=-153.718, shoulder=lefty, elbow=epositive, wrist=wpositive, fatherId=fReference[0]}
  [538] = {x=-282.882, y=194.063, rx=180, rz=-153.6, shoulder=lefty, elbow=epositive, wrist=wpositive, fatherId=fReference[0]}
  [539] = {x=-281.546, y=193.4, rx=180, rz=-153.483, shoulder=lefty, elbow=epositive, wrist=wpositive, fatherId=fReference[0]}
  [540] = {x=-280.212, y=192.734, rx=-180, rz=-153.367, shoulder=lefty, elbow=epositive, wrist=wpositive, fatherId=fReference[0]}
  [541] = {x=-278.879, y=192.066, rx=-180, rz=-153.251, shoulder=lefty, elbow=epositive, wrist=wpositive, fatherId=fReference[0]}
  [542] = {x=-277.546, y=191.394, rx=-180, rz=-153.136, shoulder=lefty, elbow=epositive, wrist=wpositive, fatherId=fReference[0]}
  [543] = {x=-276.214, y=190.719, rx=-180, rz=-153.022, shoulder=lefty, elbow=epositive, wrist=wpositive, fatherId=fReference[0]}
  [544] = {x=-274.883, y=190.042, rx=-180, rz=-152.908, shoulder=lefty, elbow=epositive, wrist=wpositive, fatherId=fReference[0]}
  [545] = {x=-273.552, y=189.361, rx=-180, rz=-152.796, shoulder=lefty, elbow=epositive, wrist=wpositive, fatherId=fReference[0]}
  [546] = {x=-272.222, y=188.678, rx=-180, rz=-152.684, shoulder=lefty, elbow=epositive, wrist=wpositive, fatherId=fReference[0]}
  [547] = {x=-270.894, y=187.991, rx=-180, rz=-152.572, shoulder=lefty, elbow=epositive, wrist=wpositive, fatherId=fReference[0]}
  [548] = {x=-269.565, y=187.302, rx=-180, rz=-152.461, shoulder=lefty, elbow=epositive, wrist=wpositive, fatherId=fReference[0]}
  [549] = {x=-268.238, y=186.61, rx=-180, rz=-152.351, shoulder=lefty, elbow=epositive, wrist=wpositive, fatherId=fReference[0]}
  [550] = {x=-266.911, y=185.915, rx=180, rz=-152.242, shoulder=lefty, elbow=epositive, wrist=wpositive, fatherId=fReference[0]}
  [551] = {x=-265.585, y=185.217, rx=180, rz=-152.134, shoulder=lefty, elbow=epositive, wrist=wpositive, fatherId=fReference[0]}
  [552] = {x=-264.26, y=184.516, rx=180, rz=-152.026, shoulder=lefty, elbow=epositive, wrist=wpositive, fatherId=fReference[0]}
  [553] = {x=-262.936, y=183.813, rx=180, rz=-151.918, shoulder=lefty, elbow=epositive, wrist=wpositive, fatherId=fReference[0]}
  [554] = {x=-261.612, y=183.107, rx=-180, rz=-151.812, shoulder=lefty, elbow=epositive, wrist=wpositive, fatherId=fReference[0]}
  [555] = {x=-260.289, y=182.398, rx=180, rz=-151.706, shoulder=lefty, elbow=epositive, wrist=wpositive, fatherId=fReference[0]}
  [556] = {x=-258.967, y=181.686, rx=180, rz=-151.601, shoulder=lefty, elbow=epositive, wrist=wpositive, fatherId=fReference[0]}
  [557] = {x=-257.646, y=180.972, rx=-180, rz=-151.496, shoulder=lefty, elbow=epositive, wrist=wpositive, fatherId=fReference[0]}
  [558] = {x=-256.325, y=180.254, rx=-180, rz=-151.392, shoulder=lefty, elbow=epositive, wrist=wpositive, fatherId=fReference[0]}
  [559] = {x=-255.005, y=179.535, rx=180, rz=-151.289, shoulder=lefty, elbow=epositive, wrist=wpositive, fatherId=fReference[0]}
  [560] = {x=-253.686, y=178.812, rx=180, rz=-151.187, shoulder=lefty, elbow=epositive, wrist=wpositive, fatherId=fReference[0]}
  [561] = {x=-252.368, y=178.087, rx=-180, rz=-151.085, shoulder=lefty, elbow=epositive, wrist=wpositive, fatherId=fReference[0]}
  [562] = {x=-251.05, y=177.359, rx=-180, rz=-150.984, shoulder=lefty, elbow=epositive, wrist=wpositive, fatherId=fReference[0]}
  [563] = {x=-249.733, y=176.629, rx=-180, rz=-150.883, shoulder=lefty, elbow=epositive, wrist=wpositive, fatherId=fReference[0]}
  [564] = {x=-248.417, y=175.895, rx=180, rz=-150.784, shoulder=lefty, elbow=epositive, wrist=wpositive, fatherId=fReference[0]}
  [565] = {x=-247.102, y=175.16, rx=180, rz=-150.685, shoulder=lefty, elbow=epositive, wrist=wpositive, fatherId=fReference[0]}
  [566] = {x=-245.787, y=174.422, rx=180, rz=-150.586, shoulder=lefty, elbow=epositive, wrist=wpositive, fatherId=fReference[0]}
  [567] = {x=-244.473, y=173.681, rx=180, rz=-150.488, shoulder=lefty, elbow=epositive, wrist=wpositive, fatherId=fReference[0]}
  [568] = {x=-243.16, y=172.937, rx=-180, rz=-150.391, shoulder=lefty, elbow=epositive, wrist=wpositive, fatherId=fReference[0]}
  [569] = {x=-241.847, y=172.192, rx=-180, rz=-150.295, shoulder=lefty, elbow=epositive, wrist=wpositive, fatherId=fReference[0]}
  [570] = {x=-240.536, y=171.443, rx=180, rz=-150.199, shoulder=lefty, elbow=epositive, wrist=wpositive, fatherId=fReference[0]}
  [571] = {x=-239.225, y=170.692, rx=180, rz=-150.104, shoulder=lefty, elbow=epositive, wrist=wpositive, fatherId=fReference[0]}
  [572] = {x=-237.914, y=169.939, rx=180, rz=-150.009, shoulder=lefty, elbow=epositive, wrist=wpositive, fatherId=fReference[0]}
  [573] = {x=-236.605, y=169.183, rx=-180, rz=-149.915, shoulder=lefty, elbow=epositive, wrist=wpositive, fatherId=fReference[0]}
  [574] = {x=-235.296, y=168.425, rx=-180, rz=-149.822, shoulder=lefty, elbow=epositive, wrist=wpositive, fatherId=fReference[0]}
  [575] = {x=-233.988, y=167.664, rx=180, rz=-149.729, shoulder=lefty, elbow=epositive, wrist=wpositive, fatherId=fReference[0]}
  [576] = {x=-232.68, y=166.901, rx=180, rz=-149.638, shoulder=lefty, elbow=epositive, wrist=wpositive, fatherId=fReference[0]}
  [577] = {x=-231.373, y=166.136, rx=180, rz=-149.546, shoulder=lefty, elbow=epositive, wrist=wpositive, fatherId=fReference[0]}
  [578] = {x=-230.067, y=165.368, rx=-180, rz=-149.456, shoulder=lefty, elbow=epositive, wrist=wpositive, fatherId=fReference[0]}
  [579] = {x=-228.762, y=164.597, rx=180, rz=-149.366, shoulder=lefty, elbow=epositive, wrist=wpositive, fatherId=fReference[0]}
  [580] = {x=-227.457, y=163.825, rx=-180, rz=-149.276, shoulder=lefty, elbow=epositive, wrist=wpositive, fatherId=fReference[0]}
  [581] = {x=-226.153, y=163.05, rx=-180, rz=-149.187, shoulder=lefty, elbow=epositive, wrist=wpositive, fatherId=fReference[0]}
  [582] = {x=-224.85, y=162.272, rx=-180, rz=-149.099, shoulder=lefty, elbow=epositive, wrist=wpositive, fatherId=fReference[0]}
  [583] = {x=-223.547, y=161.493, rx=-180, rz=-149.012, shoulder=lefty, elbow=epositive, wrist=wpositive, fatherId=fReference[0]}
  [584] = {x=-222.245, y=160.711, rx=180, rz=-148.925, shoulder=lefty, elbow=epositive, wrist=wpositive, fatherId=fReference[0]}
  [585] = {x=-220.944, y=159.927, rx=-180, rz=-148.839, shoulder=lefty, elbow=epositive, wrist=wpositive, fatherId=fReference[0]}
  [586] = {x=-219.643, y=159.14, rx=-180, rz=-148.753, shoulder=lefty, elbow=epositive, wrist=wpositive, fatherId=fReference[0]}
  [587] = {x=-218.344, y=158.351, rx=-180, rz=-148.668, shoulder=lefty, elbow=epositive, wrist=wpositive, fatherId=fReference[0]}
  [588] = {x=-217.044, y=157.56, rx=180, rz=-148.584, shoulder=lefty, elbow=epositive, wrist=wpositive, fatherId=fReference[0]}
  [589] = {x=-215.746, y=156.767, rx=-180, rz=-148.5, shoulder=lefty, elbow=epositive, wrist=wpositive, fatherId=fReference[0]}
  [590] = {x=-214.448, y=155.972, rx=-180, rz=-148.417, shoulder=lefty, elbow=epositive, wrist=wpositive, fatherId=fReference[0]}
  [591] = {x=-213.15, y=155.174, rx=180, rz=-148.334, shoulder=lefty, elbow=epositive, wrist=wpositive, fatherId=fReference[0]}
  [592] = {x=-211.854, y=154.375, rx=180, rz=-148.252, shoulder=lefty, elbow=epositive, wrist=wpositive, fatherId=fReference[0]}
  [593] = {x=-210.558, y=153.573, rx=-180, rz=-148.171, shoulder=lefty, elbow=epositive, wrist=wpositive, fatherId=fReference[0]}
  [594] = {x=-209.262, y=152.769, rx=180, rz=-148.09, shoulder=lefty, elbow=epositive, wrist=wpositive, fatherId=fReference[0]}
  [595] = {x=-207.968, y=151.962, rx=180, rz=-148.01, shoulder=lefty, elbow=epositive, wrist=wpositive, fatherId=fReference[0]}
  [596] = {x=-206.674, y=151.154, rx=-180, rz=-147.931, shoulder=lefty, elbow=epositive, wrist=wpositive, fatherId=fReference[0]}
  [597] = {x=-205.38, y=150.344, rx=180, rz=-147.852, shoulder=lefty, elbow=epositive, wrist=wpositive, fatherId=fReference[0]}
  [598] = {x=-204.088, y=149.531, rx=-180, rz=-147.774, shoulder=lefty, elbow=epositive, wrist=wpositive, fatherId=fReference[0]}
  [599] = {x=-202.795, y=148.717, rx=-180, rz=-147.696, shoulder=lefty, elbow=epositive, wrist=wpositive, fatherId=fReference[0]}
  [600] = {x=-201.504, y=147.9, rx=-180, rz=-147.619, shoulder=lefty, elbow=epositive, wrist=wpositive, fatherId=fReference[0]}
  [601] = {x=-200.213, y=147.082, rx=180, rz=-147.542, shoulder=lefty, elbow=epositive, wrist=wpositive, fatherId=fReference[0]}
  [602] = {x=-198.923, y=146.261, rx=-180, rz=-147.467, shoulder=lefty, elbow=epositive, wrist=wpositive, fatherId=fReference[0]}
  [603] = {x=-197.633, y=145.438, rx=180, rz=-147.391, shoulder=lefty, elbow=epositive, wrist=wpositive, fatherId=fReference[0]}
  [604] = {x=-196.344, y=144.614, rx=-180, rz=-147.317, shoulder=lefty, elbow=epositive, wrist=wpositive, fatherId=fReference[0]}
  [605] = {x=-195.055, y=143.787, rx=-180, rz=-147.242, shoulder=lefty, elbow=epositive, wrist=wpositive, fatherId=fReference[0]}
  [606] = {x=-193.768, y=142.958, rx=180, rz=-147.169, shoulder=lefty, elbow=epositive, wrist=wpositive, fatherId=fReference[0]}
  [607] = {x=-192.48, y=142.128, rx=180, rz=-147.096, shoulder=lefty, elbow=epositive, wrist=wpositive, fatherId=fReference[0]}
  [608] = {x=-191.194, y=141.295, rx=-180, rz=-147.024, shoulder=lefty, elbow=epositive, wrist=wpositive, fatherId=fReference[0]}
  [609] = {x=-189.908, y=140.461, rx=180, rz=-146.952, shoulder=lefty, elbow=epositive, wrist=wpositive, fatherId=fReference[0]}
  [610] = {x=-188.622, y=139.625, rx=180, rz=-146.88, shoulder=lefty, elbow=epositive, wrist=wpositive, fatherId=fReference[0]}
  [611] = {x=-187.337, y=138.786, rx=-180, rz=-146.81, shoulder=lefty, elbow=epositive, wrist=wpositive, fatherId=fReference[0]}
  [612] = {x=-186.053, y=137.946, rx=180, rz=-146.74, shoulder=lefty, elbow=epositive, wrist=wpositive, fatherId=fReference[0]}
  [613] = {x=-184.769, y=137.104, rx=180, rz=-146.67, shoulder=lefty, elbow=epositive, wrist=wpositive, fatherId=fReference[0]}
  [614] = {x=-183.486, y=136.26, rx=180, rz=-146.601, shoulder=lefty, elbow=epositive, wrist=wpositive, fatherId=fReference[0]}
  [615] = {x=-182.204, y=135.415, rx=-180, rz=-146.533, shoulder=lefty, elbow=epositive, wrist=wpositive, fatherId=fReference[0]}
  [616] = {x=-180.922, y=134.567, rx=180, rz=-146.465, shoulder=lefty, elbow=epositive, wrist=wpositive, fatherId=fReference[0]}
  [617] = {x=-179.641, y=133.718, rx=-180, rz=-146.398, shoulder=lefty, elbow=epositive, wrist=wpositive, fatherId=fReference[0]}
  [618] = {x=-178.36, y=132.867, rx=180, rz=-146.331, shoulder=lefty, elbow=epositive, wrist=wpositive, fatherId=fReference[0]}
  [619] = {x=-177.08, y=132.014, rx=180, rz=-146.265, shoulder=lefty, elbow=epositive, wrist=wpositive, fatherId=fReference[0]}
  [620] = {x=-175.8, y=131.16, rx=180, rz=-146.199, shoulder=lefty, elbow=epositive, wrist=wpositive, fatherId=fReference[0]}
  [621] = {x=-174.521, y=130.304, rx=-180, rz=-146.134, shoulder=lefty, elbow=epositive, wrist=wpositive, fatherId=fReference[0]}
  [622] = {x=-173.242, y=129.446, rx=-180, rz=-146.07, shoulder=lefty, elbow=epositive, wrist=wpositive, fatherId=fReference[0]}
  [623] = {x=-171.964, y=128.586, rx=180, rz=-146.006, shoulder=lefty, elbow=epositive, wrist=wpositive, fatherId=fReference[0]}
  [624] = {x=-170.687, y=127.724, rx=-180, rz=-145.943, shoulder=lefty, elbow=epositive, wrist=wpositive, fatherId=fReference[0]}
  [625] = {x=-169.41, y=126.861, rx=180, rz=-145.88, shoulder=lefty, elbow=epositive, wrist=wpositive, fatherId=fReference[0]}
  [626] = {x=-168.134, y=125.996, rx=180, rz=-145.818, shoulder=lefty, elbow=epositive, wrist=wpositive, fatherId=fReference[0]}
  [627] = {x=-166.858, y=125.13, rx=-180, rz=-145.756, shoulder=lefty, elbow=epositive, wrist=wpositive, fatherId=fReference[0]}
  [628] = {x=-165.583, y=124.262, rx=180, rz=-145.695, shoulder=lefty, elbow=epositive, wrist=wpositive, fatherId=fReference[0]}
  [629] = {x=-164.308, y=123.392, rx=-180, rz=-145.634, shoulder=lefty, elbow=epositive, wrist=wpositive, fatherId=fReference[0]}
  [630] = {x=-163.034, y=122.521, rx=-180, rz=-145.574, shoulder=lefty, elbow=epositive, wrist=wpositive, fatherId=fReference[0]}
  [631] = {x=-161.76, y=121.648, rx=180, rz=-145.515, shoulder=lefty, elbow=epositive, wrist=wpositive, fatherId=fReference[0]}
  [632] = {x=-160.487, y=120.773, rx=-180, rz=-145.455, shoulder=lefty, elbow=epositive, wrist=wpositive, fatherId=fReference[0]}
  [633] = {x=-159.215, y=119.897, rx=180, rz=-145.397, shoulder=lefty, elbow=epositive, wrist=wpositive, fatherId=fReference[0]}
  [634] = {x=-157.942, y=119.02, rx=-180, rz=-145.339, shoulder=lefty, elbow=epositive, wrist=wpositive, fatherId=fReference[0]}
  [635] = {x=-156.671, y=118.141, rx=-180, rz=-145.282, shoulder=lefty, elbow=epositive, wrist=wpositive, fatherId=fReference[0]}
  [636] = {x=-155.4, y=117.26, rx=-180, rz=-145.225, shoulder=lefty, elbow=epositive, wrist=wpositive, fatherId=fReference[0]}
  [637] = {x=-154.129, y=116.378, rx=180, rz=-145.168, shoulder=lefty, elbow=epositive, wrist=wpositive, fatherId=fReference[0]}
  [638] = {x=-152.859, y=115.494, rx=-180, rz=-145.113, shoulder=lefty, elbow=epositive, wrist=wpositive, fatherId=fReference[0]}
  [639] = {x=-151.59, y=114.609, rx=-180, rz=-145.057, shoulder=lefty, elbow=epositive, wrist=wpositive, fatherId=fReference[0]}
  [640] = {x=-150.321, y=113.722, rx=180, rz=-145.002, shoulder=lefty, elbow=epositive, wrist=wpositive, fatherId=fReference[0]}
  [641] = {x=-149.052, y=112.834, rx=180, rz=-144.948, shoulder=lefty, elbow=epositive, wrist=wpositive, fatherId=fReference[0]}
  [642] = {x=-147.784, y=111.944, rx=180, rz=-144.894, shoulder=lefty, elbow=epositive, wrist=wpositive, fatherId=fReference[0]}
  [643] = {x=-146.517, y=111.053, rx=180, rz=-144.841, shoulder=lefty, elbow=epositive, wrist=wpositive, fatherId=fReference[0]}
  [644] = {x=-145.25, y=110.161, rx=-180, rz=-144.789, shoulder=lefty, elbow=epositive, wrist=wpositive, fatherId=fReference[0]}
  [645] = {x=-143.983, y=109.267, rx=180, rz=-144.736, shoulder=lefty, elbow=epositive, wrist=wpositive, fatherId=fReference[0]}
  [646] = {x=-142.717, y=108.372, rx=180, rz=-144.685, shoulder=lefty, elbow=epositive, wrist=wpositive, fatherId=fReference[0]}
  [647] = {x=-141.452, y=107.475, rx=180, rz=-144.634, shoulder=lefty, elbow=epositive, wrist=wpositive, fatherId=fReference[0]}
  [648] = {x=-140.187, y=106.578, rx=180, rz=-144.583, shoulder=lefty, elbow=epositive, wrist=wpositive, fatherId=fReference[0]}
  [649] = {x=-138.922, y=105.678, rx=-180, rz=-144.533, shoulder=lefty, elbow=epositive, wrist=wpositive, fatherId=fReference[0]}
  [650] = {x=-137.658, y=104.778, rx=180, rz=-144.483, shoulder=lefty, elbow=epositive, wrist=wpositive, fatherId=fReference[0]}
  [651] = {x=-136.395, y=103.876, rx=-180, rz=-144.434, shoulder=lefty, elbow=epositive, wrist=wpositive, fatherId=fReference[0]}
  [652] = {x=-135.131, y=102.973, rx=-180, rz=-144.385, shoulder=lefty, elbow=epositive, wrist=wpositive, fatherId=fReference[0]}
  [653] = {x=-133.869, y=102.068, rx=180, rz=-144.337, shoulder=lefty, elbow=epositive, wrist=wpositive, fatherId=fReference[0]}
  [654] = {x=-132.606, y=101.162, rx=-180, rz=-144.29, shoulder=lefty, elbow=epositive, wrist=wpositive, fatherId=fReference[0]}
  [655] = {x=-131.345, y=100.255, rx=-180, rz=-144.242, shoulder=lefty, elbow=epositive, wrist=wpositive, fatherId=fReference[0]}
  [656] = {x=-130.083, y=99.347, rx=180, rz=-144.196, shoulder=lefty, elbow=epositive, wrist=wpositive, fatherId=fReference[0]}
  [657] = {x=-128.822, y=98.437, rx=180, rz=-144.15, shoulder=lefty, elbow=epositive, wrist=wpositive, fatherId=fReference[0]}
  [658] = {x=-127.562, y=97.527, rx=180, rz=-144.104, shoulder=lefty, elbow=epositive, wrist=wpositive, fatherId=fReference[0]}
  [659] = {x=-126.302, y=96.615, rx=-180, rz=-144.059, shoulder=lefty, elbow=epositive, wrist=wpositive, fatherId=fReference[0]}
  [660] = {x=-125.042, y=95.702, rx=-180, rz=-144.014, shoulder=lefty, elbow=epositive, wrist=wpositive, fatherId=fReference[0]}
  [661] = {x=-123.783, y=94.787, rx=-180, rz=-143.97, shoulder=lefty, elbow=epositive, wrist=wpositive, fatherId=fReference[0]}
  [662] = {x=-122.525, y=93.872, rx=-180, rz=-143.926, shoulder=lefty, elbow=epositive, wrist=wpositive, fatherId=fReference[0]}
  [663] = {x=-121.266, y=92.955, rx=-180, rz=-143.883, shoulder=lefty, elbow=epositive, wrist=wpositive, fatherId=fReference[0]}
  [664] = {x=-120.009, y=92.037, rx=180, rz=-143.841, shoulder=lefty, elbow=epositive, wrist=wpositive, fatherId=fReference[0]}
  [665] = {x=-118.751, y=91.118, rx=-180, rz=-143.798, shoulder=lefty, elbow=epositive, wrist=wpositive, fatherId=fReference[0]}
  [666] = {x=-117.494, y=90.198, rx=180, rz=-143.757, shoulder=lefty, elbow=epositive, wrist=wpositive, fatherId=fReference[0]}
  [667] = {x=-116.238, y=89.277, rx=180, rz=-143.715, shoulder=lefty, elbow=epositive, wrist=wpositive, fatherId=fReference[0]}
  [668] = {x=-114.981, y=88.355, rx=-180, rz=-143.675, shoulder=lefty, elbow=epositive, wrist=wpositive, fatherId=fReference[0]}
  [669] = {x=-113.726, y=87.432, rx=-180, rz=-143.634, shoulder=lefty, elbow=epositive, wrist=wpositive, fatherId=fReference[0]}
  [670] = {x=-112.47, y=86.507, rx=-180, rz=-143.595, shoulder=lefty, elbow=epositive, wrist=wpositive, fatherId=fReference[0]}
  [671] = {x=-111.215, y=85.582, rx=-180, rz=-143.555, shoulder=lefty, elbow=epositive, wrist=wpositive, fatherId=fReference[0]}
  [672] = {x=-109.961, y=84.656, rx=-180, rz=-143.516, shoulder=lefty, elbow=epositive, wrist=wpositive, fatherId=fReference[0]}
  [673] = {x=-108.707, y=83.728, rx=-180, rz=-143.478, shoulder=lefty, elbow=epositive, wrist=wpositive, fatherId=fReference[0]}
  [674] = {x=-107.453, y=82.8, rx=-180, rz=-143.44, shoulder=lefty, elbow=epositive, wrist=wpositive, fatherId=fReference[0]}
  [675] = {x=-106.2, y=81.87, rx=180, rz=-143.403, shoulder=lefty, elbow=epositive, wrist=wpositive, fatherId=fReference[0]}
  [676] = {x=-104.947, y=80.94, rx=180, rz=-143.366, shoulder=lefty, elbow=epositive, wrist=wpositive, fatherId=fReference[0]}
  [677] = {x=-103.694, y=80.008, rx=-180, rz=-143.329, shoulder=lefty, elbow=epositive, wrist=wpositive, fatherId=fReference[0]}
  [678] = {x=-102.442, y=79.076, rx=-180, rz=-143.293, shoulder=lefty, elbow=epositive, wrist=wpositive, fatherId=fReference[0]}
  [679] = {x=-101.19, y=78.143, rx=-180, rz=-143.258, shoulder=lefty, elbow=epositive, wrist=wpositive, fatherId=fReference[0]}
  [680] = {x=-99.938, y=77.208, rx=-180, rz=-143.223, shoulder=lefty, elbow=epositive, wrist=wpositive, fatherId=fReference[0]}
  [681] = {x=-98.687, y=76.273, rx=-180, rz=-143.188, shoulder=lefty, elbow=epositive, wrist=wpositive, fatherId=fReference[0]}
  [682] = {x=-97.437, y=75.337, rx=180, rz=-143.154, shoulder=lefty, elbow=epositive, wrist=wpositive, fatherId=fReference[0]}
  [683] = {x=-96.186, y=74.4, rx=-180, rz=-143.12, shoulder=lefty, elbow=epositive, wrist=wpositive, fatherId=fReference[0]}
  [684] = {x=-94.936, y=73.462, rx=180, rz=-143.087, shoulder=lefty, elbow=epositive, wrist=wpositive, fatherId=fReference[0]}
  [685] = {x=-93.686, y=72.523, rx=180, rz=-143.054, shoulder=lefty, elbow=epositive, wrist=wpositive, fatherId=fReference[0]}
  [686] = {x=-92.437, y=71.584, rx=-180, rz=-143.022, shoulder=lefty, elbow=epositive, wrist=wpositive, fatherId=fReference[0]}
  [687] = {x=-91.188, y=70.643, rx=-180, rz=-142.99, shoulder=lefty, elbow=epositive, wrist=wpositive, fatherId=fReference[0]}
  [688] = {x=-89.939, y=69.702, rx=-180, rz=-142.959, shoulder=lefty, elbow=epositive, wrist=wpositive, fatherId=fReference[0]}
  [689] = {x=-88.691, y=68.76, rx=-180, rz=-142.928, shoulder=lefty, elbow=epositive, wrist=wpositive, fatherId=fReference[0]}
  [690] = {x=-87.443, y=67.817, rx=-180, rz=-142.897, shoulder=lefty, elbow=epositive, wrist=wpositive, fatherId=fReference[0]}
  [691] = {x=-86.195, y=66.873, rx=180, rz=-142.867, shoulder=lefty, elbow=epositive, wrist=wpositive, fatherId=fReference[0]}
  [692] = {x=-84.948, y=65.929, rx=-180, rz=-142.838, shoulder=lefty, elbow=epositive, wrist=wpositive, fatherId=fReference[0]}
  [693] = {x=-83.701, y=64.984, rx=180, rz=-142.809, shoulder=lefty, elbow=epositive, wrist=wpositive, fatherId=fReference[0]}
  [694] = {x=-82.454, y=64.038, rx=180, rz=-142.78, shoulder=lefty, elbow=epositive, wrist=wpositive, fatherId=fReference[0]}
  [695] = {x=-81.208, y=63.091, rx=-180, rz=-142.752, shoulder=lefty, elbow=epositive, wrist=wpositive, fatherId=fReference[0]}
  [696] = {x=-79.962, y=62.143, rx=-180, rz=-142.724, shoulder=lefty, elbow=epositive, wrist=wpositive, fatherId=fReference[0]}
  [697] = {x=-78.716, y=61.195, rx=180, rz=-142.697, shoulder=lefty, elbow=epositive, wrist=wpositive, fatherId=fReference[0]}
  [698] = {x=-77.47, y=60.246, rx=-180, rz=-142.67, shoulder=lefty, elbow=epositive, wrist=wpositive, fatherId=fReference[0]}
  [699] = {x=-76.225, y=59.297, rx=-180, rz=-142.644, shoulder=lefty, elbow=epositive, wrist=wpositive, fatherId=fReference[0]}
  [700] = {x=-74.98, y=58.346, rx=180, rz=-142.618, shoulder=lefty, elbow=epositive, wrist=wpositive, fatherId=fReference[0]}
  [701] = {x=-73.736, y=57.395, rx=180, rz=-142.592, shoulder=lefty, elbow=epositive, wrist=wpositive, fatherId=fReference[0]}
  [702] = {x=-72.491, y=56.444, rx=-180, rz=-142.567, shoulder=lefty, elbow=epositive, wrist=wpositive, fatherId=fReference[0]}
  [703] = {x=-71.247, y=55.491, rx=-180, rz=-142.543, shoulder=lefty, elbow=epositive, wrist=wpositive, fatherId=fReference[0]}
  [704] = {x=-70.003, y=54.538, rx=180, rz=-142.518, shoulder=lefty, elbow=epositive, wrist=wpositive, fatherId=fReference[0]}
  [705] = {x=-68.76, y=53.585, rx=-180, rz=-142.495, shoulder=lefty, elbow=epositive, wrist=wpositive, fatherId=fReference[0]}
  [706] = {x=-67.516, y=52.63, rx=-180, rz=-142.471, shoulder=lefty, elbow=epositive, wrist=wpositive, fatherId=fReference[0]}
  [707] = {x=-66.273, y=51.676, rx=180, rz=-142.449, shoulder=lefty, elbow=epositive, wrist=wpositive, fatherId=fReference[0]}
  [708] = {x=-65.03, y=50.72, rx=180, rz=-142.426, shoulder=lefty, elbow=epositive, wrist=wpositive, fatherId=fReference[0]}
  [709] = {x=-63.788, y=49.764, rx=-180, rz=-142.404, shoulder=lefty, elbow=epositive, wrist=wpositive, fatherId=fReference[0]}
  [710] = {x=-62.545, y=48.808, rx=-180, rz=-142.383, shoulder=lefty, elbow=epositive, wrist=wpositive, fatherId=fReference[0]}
  [711] = {x=-61.303, y=47.85, rx=-180, rz=-142.362, shoulder=lefty, elbow=epositive, wrist=wpositive, fatherId=fReference[0]}
  [712] = {x=-60.061, y=46.893, rx=-180, rz=-142.341, shoulder=lefty, elbow=epositive, wrist=wpositive, fatherId=fReference[0]}
  [713] = {x=-58.82, y=45.934, rx=-180, rz=-142.321, shoulder=lefty, elbow=epositive, wrist=wpositive, fatherId=fReference[0]}
  [714] = {x=-57.578, y=44.976, rx=-180, rz=-142.301, shoulder=lefty, elbow=epositive, wrist=wpositive, fatherId=fReference[0]}
  [715] = {x=-56.337, y=44.016, rx=180, rz=-142.282, shoulder=lefty, elbow=epositive, wrist=wpositive, fatherId=fReference[0]}
  [716] = {x=-55.096, y=43.057, rx=180, rz=-142.263, shoulder=lefty, elbow=epositive, wrist=wpositive, fatherId=fReference[0]}
  [717] = {x=-53.855, y=42.096, rx=-180, rz=-142.244, shoulder=lefty, elbow=epositive, wrist=wpositive, fatherId=fReference[0]}
  [718] = {x=-52.615, y=41.135, rx=180, rz=-142.226, shoulder=lefty, elbow=epositive, wrist=wpositive, fatherId=fReference[0]}
  [719] = {x=-51.374, y=40.174, rx=180, rz=-142.209, shoulder=lefty, elbow=epositive, wrist=wpositive, fatherId=fReference[0]}
  [720] = {x=-50.134, y=39.212, rx=180, rz=-142.192, shoulder=lefty, elbow=epositive, wrist=wpositive, fatherId=fReference[0]}
  [721] = {x=-48.894, y=38.25, rx=-180, rz=-142.175, shoulder=lefty, elbow=epositive, wrist=wpositive, fatherId=fReference[0]}
  [722] = {x=-47.654, y=37.288, rx=-180, rz=-142.159, shoulder=lefty, elbow=epositive, wrist=wpositive, fatherId=fReference[0]}
  [723] = {x=-46.414, y=36.325, rx=-180, rz=-142.143, shoulder=lefty, elbow=epositive, wrist=wpositive, fatherId=fReference[0]}
  [724] = {x=-45.175, y=35.361, rx=180, rz=-142.127, shoulder=lefty, elbow=epositive, wrist=wpositive, fatherId=fReference[0]}
  [725] = {x=-43.935, y=34.397, rx=-180, rz=-142.112, shoulder=lefty, elbow=epositive, wrist=wpositive, fatherId=fReference[0]}
  [726] = {x=-42.696, y=33.433, rx=-180, rz=-142.098, shoulder=lefty, elbow=epositive, wrist=wpositive, fatherId=fReference[0]}
  [727] = {x=-41.457, y=32.468, rx=-180, rz=-142.083, shoulder=lefty, elbow=epositive, wrist=wpositive, fatherId=fReference[0]}
  [728] = {x=-40.218, y=31.503, rx=180, rz=-142.07, shoulder=lefty, elbow=epositive, wrist=wpositive, fatherId=fReference[0]}
  [729] = {x=-38.979, y=30.538, rx=180, rz=-142.056, shoulder=lefty, elbow=epositive, wrist=wpositive, fatherId=fReference[0]}
  [730] = {x=-37.74, y=29.572, rx=-180, rz=-142.044, shoulder=lefty, elbow=epositive, wrist=wpositive, fatherId=fReference[0]}
  [731] = {x=-36.502, y=28.606, rx=-180, rz=-142.031, shoulder=lefty, elbow=epositive, wrist=wpositive, fatherId=fReference[0]}
  [732] = {x=-35.263, y=27.639, rx=-180, rz=-142.019, shoulder=lefty, elbow=epositive, wrist=wpositive, fatherId=fReference[0]}
  [733] = {x=-34.025, y=26.672, rx=-180, rz=-142.007, shoulder=lefty, elbow=epositive, wrist=wpositive, fatherId=fReference[0]}
  [734] = {x=-32.787, y=25.705, rx=180, rz=-141.996, shoulder=lefty, elbow=epositive, wrist=wpositive, fatherId=fReference[0]}
  [735] = {x=-31.549, y=24.738, rx=-180, rz=-141.985, shoulder=lefty, elbow=epositive, wrist=wpositive, fatherId=fReference[0]}
  [736] = {x=-30.311, y=23.77, rx=-180, rz=-141.975, shoulder=lefty, elbow=epositive, wrist=wpositive, fatherId=fReference[0]}
  [737] = {x=-29.073, y=22.802, rx=-180, rz=-141.965, shoulder=lefty, elbow=epositive, wrist=wpositive, fatherId=fReference[0]}
  [738] = {x=-27.835, y=21.834, rx=-180, rz=-141.956, shoulder=lefty, elbow=epositive, wrist=wpositive, fatherId=fReference[0]}
  [739] = {x=-26.597, y=20.865, rx=-180, rz=-141.947, shoulder=lefty, elbow=epositive, wrist=wpositive, fatherId=fReference[0]}
  [740] = {x=-25.36, y=19.896, rx=180, rz=-141.938, shoulder=lefty, elbow=epositive, wrist=wpositive, fatherId=fReference[0]}
  [741] = {x=-24.122, y=18.927, rx=-180, rz=-141.93, shoulder=lefty, elbow=epositive, wrist=wpositive, fatherId=fReference[0]}
  [742] = {x=-22.885, y=17.958, rx=-180, rz=-141.922, shoulder=lefty, elbow=epositive, wrist=wpositive, fatherId=fReference[0]}
  [743] = {x=-21.647, y=16.988, rx=-180, rz=-141.915, shoulder=lefty, elbow=epositive, wrist=wpositive, fatherId=fReference[0]}
  [744] = {x=-20.41, y=16.019, rx=180, rz=-141.908, shoulder=lefty, elbow=epositive, wrist=wpositive, fatherId=fReference[0]}
  [745] = {x=-19.172, y=15.049, rx=-180, rz=-141.901, shoulder=lefty, elbow=epositive, wrist=wpositive, fatherId=fReference[0]}
  [746] = {x=-17.935, y=14.079, rx=-180, rz=-141.895, shoulder=lefty, elbow=epositive, wrist=wpositive, fatherId=fReference[0]}
  [747] = {x=-16.698, y=13.109, rx=180, rz=-141.889, shoulder=lefty, elbow=epositive, wrist=wpositive, fatherId=fReference[0]}
  [748] = {x=-15.461, y=12.138, rx=-180, rz=-141.884, shoulder=lefty, elbow=epositive, wrist=wpositive, fatherId=fReference[0]}
  [749] = {x=-14.224, y=11.168, rx=-180, rz=-141.879, shoulder=lefty, elbow=epositive, wrist=wpositive, fatherId=fReference[0]}
  [750] = {x=-12.987, y=10.197, rx=-180, rz=-141.875, shoulder=lefty, elbow=epositive, wrist=wpositive, fatherId=fReference[0]}
  [751] = {x=-11.75, y=9.226, rx=-180, rz=-141.871, shoulder=lefty, elbow=epositive, wrist=wpositive, fatherId=fReference[0]}
  [752] = {x=-10.513, y=8.255, rx=-180, rz=-141.867, shoulder=lefty, elbow=epositive, wrist=wpositive, fatherId=fReference[0]}
  [753] = {x=-9.276, y=7.284, rx=-180, rz=-141.864, shoulder=lefty, elbow=epositive, wrist=wpositive, fatherId=fReference[0]}
  [754] = {x=-8.039, y=6.313, rx=180, rz=-141.862, shoulder=lefty, elbow=epositive, wrist=wpositive, fatherId=fReference[0]}
  [755] = {x=-6.802, y=5.342, rx=180, rz=-141.859, shoulder=lefty, elbow=epositive, wrist=wpositive, fatherId=fReference[0]}
  [756] = {x=-5.565, y=4.37, rx=-180, rz=-141.857, shoulder=lefty, elbow=epositive, wrist=wpositive, fatherId=fReference[0]}
  [757] = {x=-4.328, y=3.399, rx=-180, rz=-141.856, shoulder=lefty, elbow=epositive, wrist=wpositive, fatherId=fReference[0]}
  [758] = {x=-3.091, y=2.427, rx=-180, rz=-141.855, shoulder=lefty, elbow=epositive, wrist=wpositive, fatherId=fReference[0]}
  [759] = {x=-1.854, y=1.456, rx=180, rz=-141.854, shoulder=lefty, elbow=epositive, wrist=wpositive, fatherId=fReference[0]}
  [760] = {x=-0.617, y=0.484, rx=180, rz=-141.854, shoulder=lefty, elbow=epositive, wrist=wpositive, fatherId=fReference[0]}
  [761] = {x=0.62, y=-0.487, rx=180, rz=-141.854, shoulder=lefty, elbow=epositive, wrist=wpositive, fatherId=fReference[0]}
  [762] = {x=1.857, y=-1.459, rx=-180, rz=-141.855, shoulder=lefty, elbow=epositive, wrist=wpositive, fatherId=fReference[0]}
  [763] = {x=3.094, y=-2.43, rx=-180, rz=-141.856, shoulder=lefty, elbow=epositive, wrist=wpositive, fatherId=fReference[0]}
  [764] = {x=4.331, y=-3.402, rx=-180, rz=-141.857, shoulder=lefty, elbow=epositive, wrist=wpositive, fatherId=fReference[0]}
  [765] = {x=5.568, y=-4.373, rx=-180, rz=-141.859, shoulder=lefty, elbow=epositive, wrist=wpositive, fatherId=fReference[0]}
  [766] = {x=6.805, y=-5.345, rx=180, rz=-141.862, shoulder=lefty, elbow=epositive, wrist=wpositive, fatherId=fReference[0]}
  [767] = {x=8.043, y=-6.316, rx=-180, rz=-141.864, shoulder=lefty, elbow=epositive, wrist=wpositive, fatherId=fReference[0]}
  [768] = {x=9.28, y=-7.287, rx=-180, rz=-141.867, shoulder=lefty, elbow=epositive, wrist=wpositive, fatherId=fReference[0]}
  [769] = {x=10.517, y=-8.259, rx=-180, rz=-141.871, shoulder=lefty, elbow=epositive, wrist=wpositive, fatherId=fReference[0]}
  [770] = {x=11.754, y=-9.23, rx=180, rz=-141.875, shoulder=lefty, elbow=epositive, wrist=wpositive, fatherId=fReference[0]}
  [771] = {x=12.992, y=-10.201, rx=-180, rz=-141.879, shoulder=lefty, elbow=epositive, wrist=wpositive, fatherId=fReference[0]}
  [772] = {x=14.229, y=-11.172, rx=180, rz=-141.884, shoulder=lefty, elbow=epositive, wrist=wpositive, fatherId=fReference[0]}
  [773] = {x=15.467, y=-12.143, rx=180, rz=-141.89, shoulder=lefty, elbow=epositive, wrist=wpositive, fatherId=fReference[0]}
  [774] = {x=16.704, y=-13.113, rx=180, rz=-141.895, shoulder=lefty, elbow=epositive, wrist=wpositive, fatherId=fReference[0]}
  [775] = {x=17.942, y=-14.084, rx=-180, rz=-141.901, shoulder=lefty, elbow=epositive, wrist=wpositive, fatherId=fReference[0]}
  [776] = {x=19.179, y=-15.054, rx=-180, rz=-141.908, shoulder=lefty, elbow=epositive, wrist=wpositive, fatherId=fReference[0]}
  [777] = {x=20.417, y=-16.025, rx=-180, rz=-141.915, shoulder=lefty, elbow=epositive, wrist=wpositive, fatherId=fReference[0]}
  [778] = {x=21.655, y=-16.995, rx=-180, rz=-141.922, shoulder=lefty, elbow=epositive, wrist=wpositive, fatherId=fReference[0]}
